  MoveL 657 to (55.18, -49.67, -189.83) mm, rotated rx 42.04 ry 15.1 rz 65.25 deg; joints [-16.317, -43.743, 106.759, 144.666, 49.492, -27.824, -175]
  MoveL 658 to (55.66, -49.78, -189.81) mm, rotated rx 42.04 ry 15.1 rz 65.25 deg; joints [-16.315, -43.768, 106.758, 144.655, 49.471, -27.806, -175]
  MoveL 659 to (56.16, -49.9, -189.79) mm, rotated rx 42.04 ry 15.1 rz 65.25 deg; joints [-16.314, -43.794, 106.756, 144.643, 49.448, -27.785, -175]
  MoveL 660 to (58.7, -50.57, -189.79) mm, rotated rx 42.04 ry 15.1 rz 65.25 deg; joints [-16.31, -43.921, 106.741, 144.577, 49.331, -27.679, -175]
  MoveL 661 to (60.09, -51.01, -189.88) mm, rotated rx 42.04 ry 15.1 rz 65.25 deg; joints [-16.311, -43.987, 106.725, 144.535, 49.264, -27.616, -175]
  MoveL 662 to (61.18, -51.5, -190.13) mm, rotated rx 42.04 ry 15.1 rz 65.25 deg; joints [-16.317, -44.033, 106.696, 144.49, 49.205, -27.555, -175]
  MoveL 663 to (61.98, -52.04, -190.54) mm, rotated rx 42.04 ry 15.1 rz 65.25 deg; joints [-16.329, -44.058, 106.654, 144.442, 49.153, -27.497, -175]
  MoveL 664 to (62.49, -52.65, -191.13) mm, rotated rx 42.04 ry 15.1 rz 65.25 deg; joints [-16.347, -44.062, 106.598, 144.39, 49.109, -27.442, -175]
  MoveL 665 to (62.7, -53.31, -191.87) mm, rotated rx 42.04 ry 15.1 rz 65.25 deg; joints [-16.37, -44.047, 106.53, 144.335, 49.073, -27.39, -175]
  MoveL 666 to (62.62, -54.02, -192.79) mm, rotated rx 42.04 ry 15.1 rz 65.25 deg; joints [-16.399, -44.01, 106.448, 144.277, 49.044, -27.341, -175]
  MoveL 667 to (61.57, -55.63, -195.12) mm, rotated rx 42.04 ry 15.1 rz 65.25 deg; joints [-16.475, -43.877, 106.246, 144.15, 49.009, -27.25, -175]
  MoveL 668 to (59.76, -57.01, -197.47) mm, rotated rx 42.04 ry 15.1 rz 65.25 deg; joints [-16.552, -43.706, 106.05, 144.044, 49.009, -27.192, -175]
  MoveL 669 to (57.6, -57.72, -199.17) mm, rotated rx 42.04 ry 15.1 rz 65.25 deg; joints [-16.61, -43.543, 105.918, 143.99, 49.051, -27.188, -175]
  MoveL 670 to (56.4, -57.82, -199.79) mm, rotated rx 42.04 ry 15.1 rz 65.25 deg; joints [-16.631, -43.464, 105.877, 143.983, 49.087, -27.206, -175]
  MoveL 671 to (55.1, -57.75, -200.24) mm, rotated rx 42.04 ry 15.1 rz 65.25 deg; joints [-16.648, -43.387, 105.852, 143.989, 49.134, -27.238, -175]
  MoveL 672 to (52.26, -57.11, -200.67) mm, rotated rx 42.04 ry 15.1 rz 65.25 deg; joints [-16.668, -43.239, 105.851, 144.039, 49.258, -27.343, -175]
  MoveL 673 to (51.3, -56.8, -200.71) mm, rotated rx 42.04 ry 15.1 rz 65.25 deg; joints [-16.672, -43.193, 105.861, 144.063, 49.304, -27.384, -175]
  MoveL 674 to (48.87, -55.82, -200.71) mm, rotated rx 42.04 ry 15.1 rz 65.25 deg; joints [-16.678, -43.084, 105.904, 144.132, 49.429, -27.499, -175]
  MoveL 675 to (47.92, -55.48, -200.77) mm, rotated rx 42.04 ry 15.1 rz 65.25 deg; joints [-16.683, -43.039, 105.916, 144.155, 49.476, -27.541, -175]
  MoveL 676 to (46.95, -55.09, -200.77) mm, rotated rx 42.04 ry 15.1 rz 65.25 deg; joints [-16.685, -42.995, 105.934, 144.183, 49.527, -27.587, -175]
  MoveL 677 to (46.5, -54.91, -200.78) mm, rotated rx 42.04 ry 15.1 rz 65.25 deg; joints [-16.687, -42.974, 105.941, 144.195, 49.55, -27.607, -175]
  MoveL 678 to (46.09, -54.77, -200.8) mm, rotated rx 42.04 ry 15.1 rz 65.25 deg; joints [-16.688, -42.955, 105.946, 144.205, 49.57, -27.625, -175]
  MoveL 679 to (45.66, -54.6, -200.81) mm, rotated rx 42.04 ry 15.1 rz 65.25 deg; joints [-16.69, -42.935, 105.952, 144.216, 49.592, -27.645, -175]
  MoveL 680 to (43.23, -53.62, -200.82) mm, rotated rx 42.04 ry 15.1 rz 65.25 deg; joints [-16.697, -42.825, 105.994, 144.283, 49.717, -27.758, -175]
  MoveL 681 to (42.77, -53.45, -200.83) mm, rotated rx 42.04 ry 15.1 rz 65.25 deg; joints [-16.699, -42.803, 106, 144.295, 49.74, -27.778, -175]
  MoveL 682 to (42.32, -53.31, -200.87) mm, rotated rx 42.04 ry 15.1 rz 65.25 deg; joints [-16.701, -42.781, 106.003, 144.305, 49.761, -27.797, -175]
  MoveL 683 to (41.9, -53.22, -200.91) mm, rotated rx 42.04 ry 15.1 rz 65.25 deg; joints [-16.703, -42.759, 106.003, 144.313, 49.78, -27.812, -175]
  MoveL 684 to (41.47, -53.15, -200.95) mm, rotated rx 42.04 ry 15.1 rz 65.25 deg; joints [-16.705, -42.735, 106.001, 144.321, 49.797, -27.827, -175]
  MoveL 685 to (41.03, -53.15, -200.96) mm, rotated rx 42.04 ry 15.1 rz 65.25 deg; joints [-16.705, -42.709, 105.992, 144.33, 49.811, -27.841, -175]
  MoveL 686 to (40.58, -53.2, -200.97) mm, rotated rx 42.04 ry 15.1 rz 65.25 deg; joints [-16.704, -42.682, 105.98, 144.338, 49.824, -27.852, -175]
  MoveL 687 to (41.34, -53.26, -201.71) mm, rotated rx 42.04 ry 15.1 rz 65.25 deg; joints [-16.732, -42.719, 105.975, 144.283, 49.797, -27.807, -175]
  MoveL 688 to (40.01, -53.79, -202.26) mm, rotated rx 42.04 ry 15.1 rz 65.25 deg; joints [-16.748, -42.619, 105.893, 144.273, 49.816, -27.813, -175]
  MoveL 689 to (38.53, -54.28, -202.68) mm, rotated rx 42.04 ry 15.1 rz 65.25 deg; joints [-16.759, -42.512, 105.814, 144.274, 49.841, -27.829, -175]
  MoveL 690 to (36.83, -54.75, -202.99) mm, rotated rx 42.04 ry 15.1 rz 65.25 deg; joints [-16.766, -42.394, 105.735, 144.285, 49.875, -27.856, -175]
  MoveL 691 to (34.86, -55.21, -203.17) mm, rotated rx 42.04 ry 15.1 rz 65.25 deg; joints [-16.768, -42.262, 105.654, 144.307, 49.917, -27.894, -175]
  MoveL 692 to (32.82, -55.68, -203.37) mm, rotated rx 42.04 ry 15.1 rz 65.25 deg; joints [-16.771, -42.125, 105.57, 144.331, 49.961, -27.934, -175]
  MoveL 693 to (30.73, -56.13, -203.49) mm, rotated rx 42.04 ry 15.1 rz 65.25 deg; joints [-16.77, -41.986, 105.488, 144.359, 50.007, -27.977, -175]
  MoveL 694 to (28.65, -56.6, -203.71) mm, rotated rx 42.04 ry 15.1 rz 65.25 deg; joints [-16.774, -41.847, 105.403, 144.381, 50.051, -28.016, -175]
  MoveL 695 to (26.56, -57.04, -203.83) mm, rotated rx 42.04 ry 15.1 rz 65.25 deg; joints [-16.773, -41.708, 105.321, 144.41, 50.097, -28.059, -175]
  MoveL 696 to (24.48, -57.49, -203.95) mm, rotated rx 42.04 ry 15.1 rz 65.25 deg; joints [-16.773, -41.57, 105.238, 144.437, 50.142, -28.102, -175]
  MoveL 697 to (22.39, -57.93, -204.06) mm, rotated rx 42.04 ry 15.1 rz 65.25 deg; joints [-16.772, -41.432, 105.156, 144.465, 50.188, -28.144, -175]
  MoveL 698 to (20.3, -58.38, -204.3) mm, rotated rx 42.04 ry 15.1 rz 65.25 deg; joints [-16.776, -41.292, 105.071, 144.486, 50.233, -28.183, -175]
  MoveL 699 to (18.21, -58.81, -204.42) mm, rotated rx 42.04 ry 15.1 rz 65.25 deg; joints [-16.776, -41.154, 104.988, 144.514, 50.278, -28.225, -175]
  MoveL 700 to (16.22, -59.29, -204.52) mm, rotated rx 42.04 ry 15.1 rz 65.25 deg; joints [-16.774, -41.02, 104.903, 144.539, 50.317, -28.263, -175]
  MoveL 701 to (14.29, -59.87, -204.73) mm, rotated rx 42.04 ry 15.1 rz 65.25 deg; joints [-16.776, -40.886, 104.809, 144.556, 50.35, -28.292, -175]
  MoveL 702 to (11.83, -60.35, -204.87) mm, rotated rx 42.04 ry 15.1 rz 65.25 deg; joints [-16.776, -40.724, 104.713, 144.587, 50.404, -28.342, -175]
  MoveL 703 to (9.41, -60.7, -204.95) mm, rotated rx 42.04 ry 15.1 rz 65.25 deg; joints [-16.775, -40.569, 104.63, 144.623, 50.462, -28.396, -175]
  MoveL 704 to (7.15, -61.09, -204.98) mm, rotated rx 42.04 ry 15.1 rz 65.25 deg; joints [-16.772, -40.423, 104.547, 144.658, 50.513, -28.446, -175]
  MoveL 705 to (5.14, -61.5, -205.03) mm, rotated rx 42.04 ry 15.1 rz 65.25 deg; joints [-16.769, -40.291, 104.469, 144.686, 50.556, -28.487, -175]
  MoveL 706 to (3.22, -61.89, -205.15) mm, rotated rx 42.04 ry 15.1 rz 65.25 deg; joints [-16.769, -40.164, 104.391, 144.71, 50.596, -28.524, -175]
  MoveL 707 to (1.23, -62.3, -205.21) mm, rotated rx 42.04 ry 15.1 rz 65.25 deg; joints [-16.767, -40.033, 104.311, 144.736, 50.637, -28.563, -175]
  MoveL 708 to (-0.85, -62.72, -205.28) mm, rotated rx 42.04 ry 15.1 rz 65.25 deg; joints [-16.765, -39.896, 104.227, 144.764, 50.681, -28.604, -175]
  MoveL 709 to (-2.8, -63.09, -205.46) mm, rotated rx 42.04 ry 15.1 rz 65.25 deg; joints [-16.767, -39.767, 104.148, 144.784, 50.722, -28.64, -175]
  MoveL 710 to (-4.68, -63.43, -205.78) mm, rotated rx 42.04 ry 15.1 rz 65.25 deg; joints [-16.775, -39.643, 104.071, 144.797, 50.763, -28.671, -175]
  MoveL 711 to (-5.49, -63.13, -206.82) mm, rotated rx 42.04 ry 15.1 rz 65.25 deg; joints [-16.816, -39.595, 104.059, 144.765, 50.801, -28.679, -175]
  MoveL 712 to (-5.26, -63.03, -207.34) mm, rotated rx 42.04 ry 15.1 rz 65.25 deg; joints [-16.837, -39.609, 104.063, 144.736, 50.799, -28.663, -175]
  MoveL 713 to (-5.25, -63, -207.66) mm, rotated rx 42.04 ry 15.1 rz 65.25 deg; joints [-16.849, -39.607, 104.059, 144.72, 50.8, -28.655, -175]
  MoveL 714 to (-5.46, -63.06, -207.82) mm, rotated rx 42.04 ry 15.1 rz 65.25 deg; joints [-16.855, -39.592, 104.046, 144.715, 50.804, -28.654, -175]
  MoveL 715 to (-5.84, -63.24, -207.86) mm, rotated rx 42.04 ry 15.1 rz 65.25 deg; joints [-16.854, -39.563, 104.021, 144.717, 50.806, -28.657, -175]
  MoveL 716 to (-6.28, -63.52, -207.87) mm, rotated rx 42.04 ry 15.1 rz 65.25 deg; joints [-16.852, -39.528, 103.986, 144.72, 50.806, -28.658, -175]
  MoveL 717 to (-6.74, -63.9, -207.89) mm, rotated rx 42.04 ry 15.1 rz 65.25 deg; joints [-16.849, -39.489, 103.942, 144.721, 50.802, -28.656, -175]
  MoveL 718 to (-7.21, -64.32, -207.9) mm, rotated rx 42.04 ry 15.1 rz 65.25 deg; joints [-16.846, -39.448, 103.895, 144.722, 50.795, -28.652, -175]
  MoveL 719 to (-9.77, -66.94, -207.9) mm, rotated rx 42.04 ry 15.1 rz 65.25 deg; joints [-16.823, -39.214, 103.605, 144.723, 50.745, -28.622, -175]
  MoveL 720 to (-10.09, -67.25, -207.92) mm, rotated rx 42.04 ry 15.1 rz 65.25 deg; joints [-16.822, -39.185, 103.571, 144.722, 50.74, -28.618, -175]
  MoveL 721 to (-10.43, -67.59, -207.93) mm, rotated rx 42.04 ry 15.1 rz 65.25 deg; joints [-16.819, -39.154, 103.532, 144.722, 50.733, -28.614, -175]
  MoveL 722 to (-10.8, -67.96, -207.94) mm, rotated rx 42.04 ry 15.1 rz 65.25 deg; joints [-16.816, -39.12, 103.491, 144.722, 50.726, -28.61, -175]
  MoveL 723 to (-11.16, -68.3, -207.96) mm, rotated rx 42.04 ry 15.1 rz 65.25 deg; joints [-16.814, -39.088, 103.453, 144.721, 50.72, -28.606, -175]
  MoveL 724 to (-11.5, -68.61, -208) mm, rotated rx 42.04 ry 15.1 rz 65.25 deg; joints [-16.812, -39.058, 103.416, 144.72, 50.715, -28.602, -175]
  MoveL 725 to (-11.83, -68.89, -208.06) mm, rotated rx 42.04 ry 15.1 rz 65.25 deg; joints [-16.812, -39.029, 103.383, 144.719, 50.711, -28.599, -175]
  MoveL 726 to (-12.18, -69.21, -208.09) mm, rotated rx 42.04 ry 15.1 rz 65.25 deg; joints [-16.811, -38.998, 103.346, 144.718, 50.706, -28.595, -175]
  MoveL 727 to (-12.53, -69.55, -208.11) mm, rotated rx 42.04 ry 15.1 rz 65.25 deg; joints [-16.808, -38.967, 103.308, 144.717, 50.7, -28.591, -175]
  MoveL 728 to (-12.88, -69.9, -208.11) mm, rotated rx 42.04 ry 15.1 rz 65.25 deg; joints [-16.805, -38.934, 103.268, 144.717, 50.693, -28.587, -175]
  MoveL 729 to (-13.25, -70.28, -208.11) mm, rotated rx 42.04 ry 15.1 rz 65.25 deg; joints [-16.802, -38.901, 103.227, 144.717, 50.686, -28.583, -175]
  MoveL 730 to (-15.49, -72.15, -208.46) mm, rotated rx 42.04 ry 15.1 rz 65.25 deg; joints [-16.798, -38.707, 103.002, 144.707, 50.66, -28.562, -175]
  MoveL 731 to (-16.62, -72.79, -208.89) mm, rotated rx 42.04 ry 15.1 rz 65.25 deg; joints [-16.809, -38.616, 102.911, 144.694, 50.662, -28.556, -175]
  MoveL 732 to (-17.76, -73.23, -209.5) mm, rotated rx 42.04 ry 15.1 rz 65.25 deg; joints [-16.827, -38.53, 102.834, 144.677, 50.674, -28.555, -175]
  MoveL 733 to (-20.07, -73.52, -211.23) mm, rotated rx 42.04 ry 15.1 rz 65.25 deg; joints [-16.888, -38.371, 102.72, 144.626, 50.726, -28.561, -175]
  MoveL 734 to (-22.42, -73.02, -213.65) mm, rotated rx 42.04 ry 15.1 rz 65.25 deg; joints [-16.981, -38.228, 102.662, 144.555, 50.818, -28.581, -175]
  MoveL 735 to (-24.17, -71.99, -216.08) mm, rotated rx 42.04 ry 15.1 rz 65.25 deg; joints [-17.078, -38.138, 102.663, 144.483, 50.918, -28.607, -175]
  MoveL 736 to (-24.6, -71.37, -217.03) mm, rotated rx 42.04 ry 15.1 rz 65.25 deg; joints [-17.119, -38.124, 102.689, 144.454, 50.96, -28.618, -175]
  MoveL 737 to (-24.72, -70.69, -217.81) mm, rotated rx 42.04 ry 15.1 rz 65.25 deg; joints [-17.153, -38.132, 102.731, 144.429, 50.996, -28.628, -175]
  MoveL 738 to (-24.66, -70.32, -218.13) mm, rotated rx 42.04 ry 15.1 rz 65.25 deg; joints [-17.168, -38.144, 102.759, 144.418, 51.012, -28.632, -175]
  MoveL 739 to (-24.53, -69.94, -218.41) mm, rotated rx 42.04 ry 15.1 rz 65.25 deg; joints [-17.182, -38.162, 102.79, 144.408, 51.027, -28.637, -175]
  MoveL 740 to (-24.05, -69.12, -218.84) mm, rotated rx 42.04 ry 15.1 rz 65.25 deg; joints [-17.205, -38.212, 102.865, 144.392, 51.053, -28.645, -175]
  MoveL 741 to (-23.26, -68.24, -219.1) mm, rotated rx 42.04 ry 15.1 rz 65.25 deg; joints [-17.223, -38.285, 102.957, 144.38, 51.073, -28.651, -175]
  MoveL 742 to (-22.17, -67.28, -219.19) mm, rotated rx 42.04 ry 15.1 rz 65.25 deg; joints [-17.235, -38.379, 103.065, 144.373, 51.088, -28.657, -175]
  MoveL 743 to (-21.76, -66.96, -219.19) mm, rotated rx 42.04 ry 15.1 rz 65.25 deg; joints [-17.238, -38.413, 103.104, 144.371, 51.092, -28.658, -175]
  MoveL 744 to (-21.39, -66.69, -219.16) mm, rotated rx 42.04 ry 15.1 rz 65.25 deg; joints [-17.239, -38.444, 103.137, 144.371, 51.094, -28.66, -175]
  MoveL 745 to (-21.03, -66.45, -219.12) mm, rotated rx 42.04 ry 15.1 rz 65.25 deg; joints [-17.24, -38.473, 103.167, 144.371, 51.095, -28.66, -175]
  MoveL 746 to (-20.67, -66.23, -219.06) mm, rotated rx 42.04 ry 15.1 rz 65.25 deg; joints [-17.24, -38.501, 103.197, 144.371, 51.096, -28.661, -175]
  MoveL 747 to (-20.3, -65.97, -219.02) mm, rotated rx 42.04 ry 15.1 rz 65.25 deg; joints [-17.241, -38.532, 103.229, 144.371, 51.098, -28.662, -175]
  MoveL 748 to (-19.89, -65.66, -219) mm, rotated rx 42.04 ry 15.1 rz 65.25 deg; joints [-17.243, -38.566, 103.266, 144.37, 51.101, -28.663, -175]
  MoveL 749 to (-19.48, -65.34, -219) mm, rotated rx 42.04 ry 15.1 rz 65.25 deg; joints [-17.246, -38.6, 103.304, 144.368, 51.105, -28.665, -175]
  MoveL 750 to (-19.09, -65.03, -218.99) mm, rotated rx 42.04 ry 15.1 rz 65.25 deg; joints [-17.249, -38.633, 103.341, 144.367, 51.108, -28.666, -175]
  MoveL 751 to (-18.71, -64.75, -218.97) mm, rotated rx 42.04 ry 15.1 rz 65.25 deg; joints [-17.25, -38.664, 103.375, 144.366, 51.111, -28.668, -175]
  MoveL 752 to (-18.36, -64.5, -218.92) mm, rotated rx 42.04 ry 15.1 rz 65.25 deg; joints [-17.251, -38.693, 103.405, 144.367, 51.112, -28.669, -175]
  MoveL 753 to (-18.01, -64.27, -218.86) mm, rotated rx 42.04 ry 15.1 rz 65.25 deg; joints [-17.251, -38.722, 103.435, 144.367, 51.113, -28.67, -175]
  MoveL 754 to (-17.62, -64.01, -218.8) mm, rotated rx 42.04 ry 15.1 rz 65.25 deg; joints [-17.251, -38.753, 103.469, 144.368, 51.115, -28.671, -175]
  MoveL 755 to (-17.13, -63.65, -218.77) mm, rotated rx 42.04 ry 15.1 rz 65.25 deg; joints [-17.253, -38.794, 103.513, 144.367, 51.118, -28.672, -175]
  MoveL 756 to (-16.49, -63.18, -218.75) mm, rotated rx 42.04 ry 15.1 rz 65.25 deg; joints [-17.256, -38.847, 103.569, 144.364, 51.122, -28.674, -175]
  MoveL 757 to (-15.26, -62.2, -218.75) mm, rotated rx 42.04 ry 15.1 rz 65.25 deg; joints [-17.266, -38.95, 103.683, 144.359, 51.133, -28.678, -175]
  MoveL 758 to (-14.6, -61.7, -218.71) mm, rotated rx 42.04 ry 15.1 rz 65.25 deg; joints [-17.269, -39.006, 103.744, 144.357, 51.138, -28.68, -175]
  MoveL 759 to (-14.1, -61.32, -218.7) mm, rotated rx 42.04 ry 15.1 rz 65.25 deg; joints [-17.272, -39.047, 103.789, 144.355, 51.142, -28.681, -175]
  MoveL 760 to (-13.68, -61.05, -218.7) mm, rotated rx 42.04 ry 15.1 rz 65.25 deg; joints [-17.274, -39.08, 103.822, 144.352, 51.142, -28.68, -175]
  MoveL 761 to (-13.31, -60.86, -218.67) mm, rotated rx 42.04 ry 15.1 rz 65.25 deg; joints [-17.275, -39.108, 103.848, 144.35, 51.141, -28.678, -175]
  MoveL 762 to (-13.11, -60.81, -218.57) mm, rotated rx 42.04 ry 15.1 rz 65.25 deg; joints [-17.272, -39.123, 103.859, 144.353, 51.137, -28.677, -175]
  MoveL 763 to (-13.15, -60.87, -218.35) mm, rotated rx 42.04 ry 15.1 rz 65.25 deg; joints [-17.263, -39.121, 103.857, 144.363, 51.135, -28.681, -175]
  MoveL 764 to (-13.43, -61.05, -218) mm, rotated rx 42.04 ry 15.1 rz 65.25 deg; joints [-17.248, -39.101, 103.842, 144.383, 51.135, -28.691, -175]
  MoveL 765 to (-12.78, -61.49, -217.3) mm, rotated rx 42.04 ry 15.1 rz 65.25 deg; joints [-17.219, -39.131, 103.832, 144.399, 51.095, -28.675, -175]
  MoveL 766 to (-10.78, -61.37, -217.14) mm, rotated rx 42.04 ry 15.1 rz 65.25 deg; joints [-17.215, -39.255, 103.891, 144.372, 51.041, -28.627, -175]
  MoveL 767 to (-8.86, -61.3, -216.86) mm, rotated rx 42.04 ry 15.1 rz 65.25 deg; joints [-17.207, -39.374, 103.947, 144.353, 50.988, -28.584, -175]
  MoveL 768 to (-6.93, -61.19, -216.59) mm, rotated rx 42.04 ry 15.1 rz 65.25 deg; joints [-17.198, -39.494, 104.004, 144.333, 50.935, -28.541, -175]
  MoveL 769 to (-5, -61.08, -216.32) mm, rotated rx 42.04 ry 15.1 rz 65.25 deg; joints [-17.191, -39.614, 104.062, 144.313, 50.883, -28.498, -175]
  MoveL 770 to (-2.97, -60.96, -216.1) mm, rotated rx 42.04 ry 15.1 rz 65.25 deg; joints [-17.185, -39.74, 104.121, 144.289, 50.827, -28.451, -175]
  MoveL 771 to (-0.85, -60.9, -215.96) mm, rotated rx 42.04 ry 15.1 rz 65.25 deg; joints [-17.181, -39.868, 104.176, 144.258, 50.767, -28.396, -175]
  MoveL 772 to (1.68, -60.93, -215.85) mm, rotated rx 42.04 ry 15.1 rz 65.25 deg; joints [-17.179, -40.018, 104.23, 144.215, 50.688, -28.325, -175]
  MoveL 773 to (4.15, -60.61, -215.78) mm, rotated rx 42.04 ry 15.1 rz 65.25 deg; joints [-17.18, -40.175, 104.313, 144.178, 50.629, -28.269, -175]
  MoveL 774 to (6.25, -60.33, -215.66) mm, rotated rx 42.04 ry 15.1 rz 65.25 deg; joints [-17.179, -40.309, 104.384, 144.148, 50.578, -28.222, -175]
  MoveL 775 to (8.13, -60.14, -215.48) mm, rotated rx 42.04 ry 15.1 rz 65.25 deg; joints [-17.176, -40.428, 104.445, 144.125, 50.529, -28.179, -175]
  MoveL 776 to (10.16, -59.96, -215.36) mm, rotated rx 42.04 ry 15.1 rz 65.25 deg; joints [-17.174, -40.554, 104.505, 144.095, 50.475, -28.13, -175]
  MoveL 777 to (12.24, -59.79, -215.22) mm, rotated rx 42.04 ry 15.1 rz 65.25 deg; joints [-17.171, -40.683, 104.566, 144.065, 50.419, -28.079, -175]
  MoveL 778 to (14.4, -59.62, -215.16) mm, rotated rx 42.04 ry 15.1 rz 65.25 deg; joints [-17.172, -40.817, 104.627, 144.029, 50.361, -28.023, -175]
  MoveL 779 to (16.53, -59.44, -214.93) mm, rotated rx 42.04 ry 15.1 rz 65.25 deg; joints [-17.166, -40.95, 104.691, 144.002, 50.303, -27.973, -175]
  MoveL 780 to (18.66, -59.26, -214.82) mm, rotated rx 42.04 ry 15.1 rz 65.25 deg; joints [-17.165, -41.082, 104.752, 143.969, 50.245, -27.919, -175]
  MoveL 781 to (20.78, -59.07, -214.6) mm, rotated rx 42.04 ry 15.1 rz 65.25 deg; joints [-17.159, -41.216, 104.816, 143.942, 50.188, -27.869, -175]
  MoveL 782 to (22.91, -58.88, -214.49) mm, rotated rx 42.04 ry 15.1 rz 65.25 deg; joints [-17.158, -41.348, 104.877, 143.908, 50.13, -27.815, -175]
  MoveL 783 to (25.04, -58.68, -214.27) mm, rotated rx 42.04 ry 15.1 rz 65.25 deg; joints [-17.153, -41.481, 104.942, 143.88, 50.073, -27.764, -175]
  MoveL 784 to (27.16, -58.49, -214.16) mm, rotated rx 42.04 ry 15.1 rz 65.25 deg; joints [-17.152, -41.613, 105.002, 143.846, 50.015, -27.71, -175]
  MoveL 785 to (29.29, -58.3, -214.05) mm, rotated rx 42.04 ry 15.1 rz 65.25 deg; joints [-17.151, -41.745, 105.062, 143.812, 49.957, -27.655, -175]
  MoveL 786 to (31.19, -58.06, -213.82) mm, rotated rx 42.04 ry 15.1 rz 65.25 deg; joints [-17.145, -41.866, 105.124, 143.789, 49.907, -27.612, -175]
  MoveL 787 to (33, -57.8, -213.52) mm, rotated rx 42.04 ry 15.1 rz 65.25 deg; joints [-17.137, -41.984, 105.188, 143.772, 49.862, -27.574, -175]
  MoveL 788 to (34.78, -57.5, -213.13) mm, rotated rx 42.04 ry 15.1 rz 65.25 deg; joints [-17.126, -42.101, 105.256, 143.761, 49.819, -27.541, -175]
  MoveL 789 to (33.37, -57.33, -212.2) mm, rotated rx 42.04 ry 15.1 rz 65.25 deg; joints [-17.092, -42.031, 105.262, 143.84, 49.871, -27.616, -175]
  MoveL 790 to (33.73, -57.31, -212.15) mm, rotated rx 42.04 ry 15.1 rz 65.25 deg; joints [-17.09, -42.054, 105.272, 143.836, 49.861, -27.607, -175]
  MoveL 791 to (34.1, -57.32, -212.09) mm, rotated rx 42.04 ry 15.1 rz 65.25 deg; joints [-17.088, -42.076, 105.279, 143.831, 49.848, -27.597, -175]
  MoveL 792 to (34.51, -57.41, -212.06) mm, rotated rx 42.04 ry 15.1 rz 65.25 deg; joints [-17.086, -42.097, 105.28, 143.823, 49.831, -27.582, -175]
  MoveL 793 to (34.93, -57.56, -212.03) mm, rotated rx 42.04 ry 15.1 rz 65.25 deg; joints [-17.084, -42.117, 105.275, 143.812, 49.811, -27.564, -175]
  MoveL 794 to (35.39, -57.78, -212.03) mm, rotated rx 42.04 ry 15.1 rz 65.25 deg; joints [-17.082, -42.137, 105.264, 143.8, 49.786, -27.541, -175]
  MoveL 795 to (35.84, -58.02, -212.02) mm, rotated rx 42.04 ry 15.1 rz 65.25 deg; joints [-17.08, -42.155, 105.252, 143.786, 49.76, -27.518, -175]
  MoveL 796 to (36.76, -58.54, -212.02) mm, rotated rx 42.04 ry 15.1 rz 65.25 deg; joints [-17.077, -42.192, 105.224, 143.758, 49.706, -27.469, -175]
  MoveL 797 to (37.19, -58.76, -212) mm, rotated rx 42.04 ry 15.1 rz 65.25 deg; joints [-17.074, -42.21, 105.212, 143.746, 49.682, -27.447, -175]
  MoveL 798 to (37.62, -58.96, -211.95) mm, rotated rx 42.04 ry 15.1 rz 65.25 deg; joints [-17.071, -42.229, 105.204, 143.736, 49.659, -27.428, -175]
  MoveL 799 to (38.1, -59.17, -211.88) mm, rotated rx 42.04 ry 15.1 rz 65.25 deg; joints [-17.067, -42.251, 105.196, 143.727, 49.634, -27.407, -175]
  MoveL 800 to (38.62, -59.42, -211.81) mm, rotated rx 42.04 ry 15.1 rz 65.25 deg; joints [-17.063, -42.274, 105.185, 143.715, 49.605, -27.383, -175]
  MoveL 801 to (39.13, -59.68, -211.78) mm, rotated rx 42.04 ry 15.1 rz 65.25 deg; joints [-17.059, -42.295, 105.172, 143.701, 49.577, -27.357, -175]
  MoveL 802 to (39.61, -59.94, -211.77) mm, rotated rx 42.04 ry 15.1 rz 65.25 deg; joints [-17.057, -42.315, 105.158, 143.687, 49.55, -27.333, -175]
  MoveL 803 to (40.07, -60.2, -211.76) mm, rotated rx 42.04 ry 15.1 rz 65.25 deg; joints [-17.055, -42.333, 105.144, 143.673, 49.522, -27.308, -175]
  MoveL 804 to (40.99, -60.71, -211.76) mm, rotated rx 42.04 ry 15.1 rz 65.25 deg; joints [-17.051, -42.37, 105.115, 143.644, 49.469, -27.259, -175]
  MoveL 805 to (41.9, -61.19, -211.74) mm, rotated rx 42.04 ry 15.1 rz 65.25 deg; joints [-17.047, -42.408, 105.091, 143.618, 49.418, -27.213, -175]
  MoveL 806 to (44.19, -62.47, -211.74) mm, rotated rx 42.04 ry 15.1 rz 65.25 deg; joints [-17.038, -42.498, 105.019, 143.546, 49.285, -27.09, -175]
  MoveL 807 to (45.41, -63.23, -211.83) mm, rotated rx 42.04 ry 15.1 rz 65.25 deg; joints [-17.036, -42.543, 104.972, 143.502, 49.21, -27.019, -175]
  MoveL 808 to (46.33, -63.98, -212.09) mm, rotated rx 42.04 ry 15.1 rz 65.25 deg; joints [-17.04, -42.569, 104.917, 143.455, 49.146, -26.953, -175]
  MoveL 809 to (46.93, -64.7, -212.53) mm, rotated rx 42.04 ry 15.1 rz 65.25 deg; joints [-17.051, -42.576, 104.855, 143.407, 49.094, -26.893, -175]
  MoveL 810 to (47.11, -65.05, -212.81) mm, rotated rx 42.04 ry 15.1 rz 65.25 deg; joints [-17.059, -42.573, 104.821, 143.381, 49.072, -26.866, -175]
  MoveL 811 to (47.22, -65.4, -213.14) mm, rotated rx 42.04 ry 15.1 rz 65.25 deg; joints [-17.068, -42.564, 104.786, 143.356, 49.053, -26.84, -175]
  MoveL 812 to (47.19, -66.08, -213.93) mm, rotated rx 42.04 ry 15.1 rz 65.25 deg; joints [-17.092, -42.533, 104.709, 143.303, 49.023, -26.792, -175]
  MoveL 813 to (46.85, -66.74, -214.9) mm, rotated rx 42.04 ry 15.1 rz 65.25 deg; joints [-17.123, -42.483, 104.625, 143.249, 49.004, -26.75, -175]
  MoveL 814 to (45.24, -68, -217.35) mm, rotated rx 42.04 ry 15.1 rz 65.25 deg; joints [-17.203, -42.326, 104.435, 143.134, 49, -26.684, -175]
  MoveL 815 to (42.96, -68.83, -219.81) mm, rotated rx 42.04 ry 15.1 rz 65.25 deg; joints [-17.287, -42.145, 104.271, 143.042, 49.037, -26.656, -175]
  MoveL 816 to (40.6, -68.88, -221.56) mm, rotated rx 42.04 ry 15.1 rz 65.25 deg; joints [-17.351, -41.991, 104.187, 143.001, 49.111, -26.68, -175]
  MoveL 817 to (39.39, -68.61, -222.18) mm, rotated rx 42.04 ry 15.1 rz 65.25 deg; joints [-17.375, -41.925, 104.176, 143.001, 49.162, -26.712, -175]
  MoveL 818 to (38.16, -68.16, -222.61) mm, rotated rx 42.04 ry 15.1 rz 65.25 deg; joints [-17.394, -41.865, 104.185, 143.013, 49.222, -26.757, -175]
  MoveL 819 to (35.64, -66.66, -222.97) mm, rotated rx 42.04 ry 15.1 rz 65.25 deg; joints [-17.419, -41.766, 104.263, 143.076, 49.371, -26.886, -175]
  MoveL 820 to (33.52, -65.1, -222.96) mm, rotated rx 42.04 ry 15.1 rz 65.25 deg; joints [-17.431, -41.694, 104.362, 143.148, 49.51, -27.014, -175]
  MoveL 821 to (33.1, -64.78, -222.95) mm, rotated rx 42.04 ry 15.1 rz 65.25 deg; joints [-17.433, -41.68, 104.382, 143.164, 49.538, -27.041, -175]
  MoveL 822 to (32.68, -64.44, -222.92) mm, rotated rx 42.04 ry 15.1 rz 65.25 deg; joints [-17.434, -41.667, 104.405, 143.18, 49.567, -27.068, -175]
  MoveL 823 to (32.28, -64.14, -222.91) mm, rotated rx 42.04 ry 15.1 rz 65.25 deg; joints [-17.436, -41.654, 104.424, 143.194, 49.594, -27.093, -175]
  MoveL 824 to (31.92, -63.89, -222.93) mm, rotated rx 42.04 ry 15.1 rz 65.25 deg; joints [-17.439, -41.641, 104.439, 143.205, 49.617, -27.113, -175]
  MoveL 825 to (31.52, -63.61, -222.96) mm, rotated rx 42.04 ry 15.1 rz 65.25 deg; joints [-17.442, -41.626, 104.456, 143.217, 49.643, -27.136, -175]
  MoveL 826 to (31.03, -63.3, -223.02) mm, rotated rx 42.04 ry 15.1 rz 65.25 deg; joints [-17.447, -41.607, 104.472, 143.23, 49.673, -27.162, -175]
  MoveL 827 to (30.53, -63, -223.1) mm, rotated rx 42.04 ry 15.1 rz 65.25 deg; joints [-17.452, -41.588, 104.487, 143.241, 49.702, -27.187, -175]
  MoveL 828 to (30.06, -62.69, -223.15) mm, rotated rx 42.04 ry 15.1 rz 65.25 deg; joints [-17.456, -41.57, 104.505, 143.254, 49.731, -27.212, -175]
  MoveL 829 to (29.62, -62.39, -223.18) mm, rotated rx 42.04 ry 15.1 rz 65.25 deg; joints [-17.459, -41.554, 104.522, 143.267, 49.759, -27.237, -175]
  MoveL 830 to (29.2, -62.09, -223.19) mm, rotated rx 42.04 ry 15.1 rz 65.25 deg; joints [-17.462, -41.539, 104.541, 143.281, 49.787, -27.262, -175]
  MoveL 831 to (28.78, -61.78, -223.19) mm, rotated rx 42.04 ry 15.1 rz 65.25 deg; joints [-17.464, -41.525, 104.56, 143.295, 49.814, -27.287, -175]
  MoveL 832 to (28.31, -61.46, -223.22) mm, rotated rx 42.04 ry 15.1 rz 65.25 deg; joints [-17.468, -41.507, 104.578, 143.309, 49.844, -27.313, -175]
  MoveL 833 to (27.84, -61.17, -223.27) mm, rotated rx 42.04 ry 15.1 rz 65.25 deg; joints [-17.472, -41.489, 104.594, 143.321, 49.872, -27.338, -175]
  MoveL 834 to (27.35, -60.89, -223.34) mm, rotated rx 42.04 ry 15.1 rz 65.25 deg; joints [-17.477, -41.469, 104.607, 143.332, 49.9, -27.362, -175]
  MoveL 835 to (26.89, -60.69, -223.4) mm, rotated rx 42.04 ry 15.1 rz 65.25 deg; joints [-17.48, -41.448, 104.615, 143.342, 49.924, -27.383, -175]
  MoveL 836 to (26.45, -60.54, -223.43) mm, rotated rx 42.04 ry 15.1 rz 65.25 deg; joints [-17.483, -41.427, 104.619, 143.352, 49.945, -27.401, -175]
  MoveL 837 to (26.06, -60.48, -223.44) mm, rotated rx 42.04 ry 15.1 rz 65.25 deg; joints [-17.483, -41.406, 104.617, 143.361, 49.96, -27.416, -175]
  MoveL 838 to (25.67, -60.44, -223.44) mm, rotated rx 42.04 ry 15.1 rz 65.25 deg; joints [-17.483, -41.384, 104.612, 143.369, 49.974, -27.429, -175]
  MoveL 839 to (26.93, -60.72, -224.32) mm, rotated rx 42.04 ry 15.1 rz 65.25 deg; joints [-17.515, -41.441, 104.595, 143.294, 49.922, -27.355, -175]
  MoveL 840 to (25.33, -60.76, -224.6) mm, rotated rx 42.04 ry 15.1 rz 65.25 deg; joints [-17.524, -41.344, 104.554, 143.312, 49.97, -27.395, -175]
  MoveL 841 to (23.52, -60.76, -224.79) mm, rotated rx 42.04 ry 15.1 rz 65.25 deg; joints [-17.53, -41.236, 104.514, 143.338, 50.026, -27.446, -175]
  MoveL 842 to (21.47, -60.71, -224.92) mm, rotated rx 42.04 ry 15.1 rz 65.25 deg; joints [-17.534, -41.117, 104.475, 143.374, 50.092, -27.507, -175]
  MoveL 843 to (19.22, -60.62, -225.01) mm, rotated rx 42.04 ry 15.1 rz 65.25 deg; joints [-17.537, -40.987, 104.436, 143.416, 50.166, -27.576, -175]
  MoveL 844 to (17.09, -60.56, -225.16) mm, rotated rx 42.04 ry 15.1 rz 65.25 deg; joints [-17.541, -40.862, 104.395, 143.452, 50.234, -27.639, -175]
  MoveL 845 to (14.95, -60.51, -225.37) mm, rotated rx 42.04 ry 15.1 rz 65.25 deg; joints [-17.548, -40.736, 104.352, 143.485, 50.303, -27.699, -175]
  MoveL 846 to (12.93, -60.44, -225.5) mm, rotated rx 42.04 ry 15.1 rz 65.25 deg; joints [-17.552, -40.618, 104.314, 143.519, 50.368, -27.759, -175]
  MoveL 847 to (11.08, -60.4, -225.76) mm, rotated rx 42.04 ry 15.1 rz 65.25 deg; joints [-17.561, -40.508, 104.273, 143.543, 50.426, -27.809, -175]
  MoveL 848 to (9.01, -60.34, -225.98) mm, rotated rx 42.04 ry 15.1 rz 65.25 deg; joints [-17.568, -40.387, 104.231, 143.573, 50.492, -27.867, -175]
  MoveL 849 to (6.93, -60.26, -226.12) mm, rotated rx 42.04 ry 15.1 rz 65.25 deg; joints [-17.573, -40.265, 104.192, 143.608, 50.559, -27.928, -175]
  MoveL 850 to (4.8, -60.17, -226.22) mm, rotated rx 42.04 ry 15.1 rz 65.25 deg; joints [-17.576, -40.141, 104.152, 143.645, 50.628, -27.991, -175]
  MoveL 851 to (2.68, -60.09, -226.45) mm, rotated rx 42.04 ry 15.1 rz 65.25 deg; joints [-17.584, -40.016, 104.109, 143.676, 50.696, -28.05, -175]
  MoveL 852 to (0.53, -59.98, -226.71) mm, rotated rx 42.04 ry 15.1 rz 65.25 deg; joints [-17.593, -39.891, 104.067, 143.705, 50.765, -28.11, -175]
  MoveL 853 to (-1.59, -59.88, -226.8) mm, rotated rx 42.04 ry 15.1 rz 65.25 deg; joints [-17.596, -39.768, 104.028, 143.742, 50.834, -28.172, -175]
  MoveL 854 to (-3.76, -59.78, -226.84) mm, rotated rx 42.04 ry 15.1 rz 65.25 deg; joints [-17.597, -39.642, 103.988, 143.783, 50.904, -28.238, -175]
  MoveL 855 to (-5.87, -59.68, -226.95) mm, rotated rx 42.04 ry 15.1 rz 65.25 deg; joints [-17.6, -39.519, 103.949, 143.818, 50.972, -28.299, -175]
  MoveL 856 to (-7.99, -59.57, -227.15) mm, rotated rx 42.04 ry 15.1 rz 65.25 deg; joints [-17.608, -39.396, 103.908, 143.849, 51.04, -28.359, -175]
  MoveL 857 to (-10.06, -59.44, -227.48) mm, rotated rx 42.04 ry 15.1 rz 65.25 deg; joints [-17.62, -39.274, 103.865, 143.873, 51.107, -28.413, -175]
  MoveL 858 to (-12.21, -59.29, -227.74) mm, rotated rx 42.04 ry 15.1 rz 65.25 deg; joints [-17.629, -39.149, 103.824, 143.902, 51.178, -28.473, -175]
  MoveL 859 to (-14.34, -59.15, -227.94) mm, rotated rx 42.04 ry 15.1 rz 65.25 deg; joints [-17.637, -39.025, 103.785, 143.933, 51.247, -28.533, -175]
  MoveL 860 to (-16.51, -58.99, -228.18) mm, rotated rx 42.04 ry 15.1 rz 65.25 deg; joints [-17.645, -38.899, 103.744, 143.962, 51.319, -28.594, -175]
  MoveL 861 to (-18.66, -58.86, -228.32) mm, rotated rx 42.04 ry 15.1 rz 65.25 deg; joints [-17.65, -38.774, 103.703, 143.996, 51.388, -28.655, -175]
  MoveL 862 to (-20.77, -58.76, -228.34) mm, rotated rx 42.04 ry 15.1 rz 65.25 deg; joints [-17.651, -38.651, 103.662, 144.034, 51.454, -28.717, -175]
  MoveL 863 to (-21.27, -58.36, -229.01) mm, rotated rx 42.04 ry 15.1 rz 65.25 deg; joints [-17.679, -38.628, 103.671, 144.016, 51.487, -28.729, -175]
  MoveL 864 to (-20.95, -58.29, -229.34) mm, rotated rx 42.04 ry 15.1 rz 65.25 deg; joints [-17.692, -38.646, 103.678, 143.995, 51.481, -28.714, -175]
  MoveL 865 to (-20.91, -58.28, -229.55) mm, rotated rx 42.04 ry 15.1 rz 65.25 deg; joints [-17.7, -38.648, 103.676, 143.984, 51.481, -28.708, -175]
  MoveL 866 to (-21.12, -58.32, -229.65) mm, rotated rx 42.04 ry 15.1 rz 65.25 deg; joints [-17.703, -38.633, 103.666, 143.982, 51.485, -28.71, -175]
  MoveL 867 to (-21.52, -58.46, -229.67) mm, rotated rx 42.04 ry 15.1 rz 65.25 deg; joints [-17.702, -38.605, 103.643, 143.986, 51.49, -28.715, -175]
  MoveC 868 to (-22.42, -58.93, -229.67) mm, rotated rx 42.04 ry 15.1 rz 65.25 deg; joints [-17.698, -38.536, 103.581, 143.994, 51.493, -28.721, -175] to (-23.29, -59.45, -229.67) mm, rotated rx 42.04 ry 15.1 rz 65.25 deg; joints [-17.692, -38.469, 103.514, 144.001, 51.493, -28.724, -175]
  MoveL 869 to (-23.29, -59.45, -229.67) mm, rotated rx 42.04 ry 15.1 rz 65.25 deg; joints [-17.693, -38.468, 103.514, 144.001, 51.493, -28.724, -175]
  MoveL 870 to (-23.76, -59.72, -229.69) mm, rotated rx 42.04 ry 15.1 rz 65.25 deg; joints [-17.691, -38.432, 103.479, 144.004, 51.493, -28.726, -175]
  MoveL 871 to (-24.24, -59.98, -229.74) mm, rotated rx 42.04 ry 15.1 rz 65.25 deg; joints [-17.69, -38.395, 103.444, 144.005, 51.494, -28.727, -175]
  MoveL 872 to (-24.76, -60.24, -229.81) mm, rotated rx 42.04 ry 15.1 rz 65.25 deg; joints [-17.69, -38.356, 103.407, 144.007, 51.497, -28.729, -175]
  MoveL 873 to (-25.28, -60.53, -229.85) mm, rotated rx 42.04 ry 15.1 rz 65.25 deg; joints [-17.689, -38.316, 103.369, 144.009, 51.498, -28.731, -175]
  MoveL 874 to (-26.33, -61.14, -229.88) mm, rotated rx 42.04 ry 15.1 rz 65.25 deg; joints [-17.683, -38.234, 103.289, 144.016, 51.498, -28.735, -175]
  MoveL 875 to (-26.81, -61.41, -229.91) mm, rotated rx 42.04 ry 15.1 rz 65.25 deg; joints [-17.682, -38.197, 103.253, 144.019, 51.499, -28.737, -175]
  MoveL 876 to (-27.24, -61.61, -229.98) mm, rotated rx 42.04 ry 15.1 rz 65.25 deg; joints [-17.683, -38.164, 103.224, 144.019, 51.501, -28.739, -175]
  MoveL 877 to (-27.64, -61.79, -230.07) mm, rotated rx 42.04 ry 15.1 rz 65.25 deg; joints [-17.684, -38.134, 103.197, 144.019, 51.504, -28.74, -175]
  MoveL 878 to (-28.02, -61.98, -230.13) mm, rotated rx 42.04 ry 15.1 rz 65.25 deg; joints [-17.685, -38.105, 103.17, 144.019, 51.506, -28.742, -175]
  MoveL 879 to (-28.42, -62.19, -230.17) mm, rotated rx 42.04 ry 15.1 rz 65.25 deg; joints [-17.684, -38.075, 103.141, 144.02, 51.507, -28.743, -175]
  MoveL 880 to (-30.66, -63.55, -230.17) mm, rotated rx 42.04 ry 15.1 rz 65.25 deg; joints [-17.671, -37.9, 102.967, 144.037, 51.504, -28.749, -175]
  MoveL 881 to (-33.27, -64.82, -230.52) mm, rotated rx 42.04 ry 15.1 rz 65.25 deg; joints [-17.671, -37.702, 102.784, 144.043, 51.516, -28.76, -175]
  MoveL 882 to (-34.51, -65.18, -230.95) mm, rotated rx 42.04 ry 15.1 rz 65.25 deg; joints [-17.683, -37.614, 102.713, 144.037, 51.533, -28.768, -175]
  MoveL 883 to (-35.69, -65.34, -231.55) mm, rotated rx 42.04 ry 15.1 rz 65.25 deg; joints [-17.703, -37.534, 102.657, 144.025, 51.558, -28.778, -175]
  MoveL 884 to (-36.83, -65.31, -232.33) mm, rotated rx 42.04 ry 15.1 rz 65.25 deg; joints [-17.731, -37.461, 102.615, 144.006, 51.59, -28.789, -175]
  MoveL 885 to (-37.91, -65.1, -233.27) mm, rotated rx 42.04 ry 15.1 rz 65.25 deg; joints [-17.768, -37.395, 102.587, 143.981, 51.63, -28.802, -175]
  MoveL 886 to (-39.94, -64.1, -235.69) mm, rotated rx 42.04 ry 15.1 rz 65.25 deg; joints [-17.865, -37.284, 102.574, 143.912, 51.733, -28.833, -175]
  MoveL 887 to (-41.27, -62.73, -238.1) mm, rotated rx 42.04 ry 15.1 rz 65.25 deg; joints [-17.966, -37.226, 102.61, 143.837, 51.833, -28.86, -175]
  MoveL 888 to (-41.48, -62.06, -239.05) mm, rotated rx 42.04 ry 15.1 rz 65.25 deg; joints [-18.007, -37.226, 102.644, 143.805, 51.871, -28.868, -175]
  MoveL 889 to (-41.39, -61.38, -239.83) mm, rotated rx 42.04 ry 15.1 rz 65.25 deg; joints [-18.041, -37.246, 102.689, 143.776, 51.9, -28.872, -175]
  MoveL 890 to (-41.23, -61.05, -240.15) mm, rotated rx 42.04 ry 15.1 rz 65.25 deg; joints [-18.057, -37.262, 102.715, 143.763, 51.911, -28.873, -175]
  MoveL 891 to (-40.99, -60.72, -240.43) mm, rotated rx 42.04 ry 15.1 rz 65.25 deg; joints [-18.07, -37.284, 102.744, 143.75, 51.921, -28.873, -175]
  MoveL 892 to (-40.3, -60.05, -240.86) mm, rotated rx 42.04 ry 15.1 rz 65.25 deg; joints [-18.093, -37.342, 102.811, 143.728, 51.933, -28.87, -175]
  MoveL 893 to (-39.31, -59.39, -241.12) mm, rotated rx 42.04 ry 15.1 rz 65.25 deg; joints [-18.109, -37.419, 102.888, 143.709, 51.937, -28.863, -175]
  MoveL 894 to (-38.01, -58.73, -241.21) mm, rotated rx 42.04 ry 15.1 rz 65.25 deg; joints [-18.119, -37.516, 102.976, 143.693, 51.933, -28.852, -175]
  MoveL 895 to (-37.53, -58.52, -241.21) mm, rotated rx 42.04 ry 15.1 rz 65.25 deg; joints [-18.121, -37.551, 103.007, 143.689, 51.93, -28.848, -175]
  MoveL 896 to (-37.12, -58.35, -241.17) mm, rotated rx 42.04 ry 15.1 rz 65.25 deg; joints [-18.122, -37.581, 103.033, 143.686, 51.926, -28.844, -175]
  MoveL 897 to (-36.72, -58.21, -241.12) mm, rotated rx 42.04 ry 15.1 rz 65.25 deg; joints [-18.121, -37.609, 103.056, 143.684, 51.922, -28.841, -175]
  MoveL 898 to (-36.33, -58.09, -241.05) mm, rotated rx 42.04 ry 15.1 rz 65.25 deg; joints [-18.12, -37.637, 103.078, 143.683, 51.917, -28.837, -175]
  MoveL 899 to (-35.92, -57.93, -241) mm, rotated rx 42.04 ry 15.1 rz 65.25 deg; joints [-18.12, -37.667, 103.103, 143.681, 51.913, -28.833, -175]
  MoveL 900 to (-35.45, -57.73, -240.98) mm, rotated rx 42.04 ry 15.1 rz 65.25 deg; joints [-18.121, -37.701, 103.132, 143.677, 51.91, -28.829, -175]
  MoveL 901 to (-30.23, -55.38, -240.97) mm, rotated rx 42.04 ry 15.1 rz 65.25 deg; joints [-18.146, -38.084, 103.466, 143.625, 51.876, -28.782, -175]
  MoveL 902 to (-29.53, -55.08, -240.96) mm, rotated rx 42.04 ry 15.1 rz 65.25 deg; joints [-18.149, -38.136, 103.51, 143.618, 51.871, -28.775, -175]
  MoveL 903 to (-28.91, -54.84, -240.95) mm, rotated rx 42.04 ry 15.1 rz 65.25 deg; joints [-18.151, -38.179, 103.545, 143.612, 51.865, -28.767, -175]
  MoveL 904 to (-28.35, -54.72, -240.94) mm, rotated rx 42.04 ry 15.1 rz 65.25 deg; joints [-18.152, -38.217, 103.57, 143.604, 51.854, -28.757, -175]
  MoveL 905 to (-27.81, -54.68, -240.9) mm, rotated rx 42.04 ry 15.1 rz 65.25 deg; joints [-18.151, -38.251, 103.587, 143.598, 51.841, -28.745, -175]
  MoveL 906 to (-27.48, -54.71, -240.74) mm, rotated rx 42.04 ry 15.1 rz 65.25 deg; joints [-18.145, -38.271, 103.595, 143.599, 51.83, -28.739, -175]
  MoveL 907 to (-27.48, -54.74, -240.43) mm, rotated rx 42.04 ry 15.1 rz 65.25 deg; joints [-18.133, -38.272, 103.6, 143.614, 51.829, -28.746, -175]
  MoveL 908 to (-27.85, -54.75, -239.94) mm, rotated rx 42.04 ry 15.1 rz 65.25 deg; joints [-18.115, -38.254, 103.6, 143.645, 51.84, -28.768, -175]
  MoveL 909 to (-27.62, -55.34, -238.97) mm, rotated rx 42.04 ry 15.1 rz 65.25 deg; joints [-18.073, -38.258, 103.576, 143.68, 51.806, -28.764, -175]
  MoveL 910 to (-25.78, -55.69, -238.67) mm, rotated rx 42.04 ry 15.1 rz 65.25 deg; joints [-18.06, -38.36, 103.595, 143.657, 51.737, -28.707, -175]
  MoveL 911 to (-23.85, -56.05, -238.46) mm, rotated rx 42.04 ry 15.1 rz 65.25 deg; joints [-18.051, -38.466, 103.614, 143.627, 51.664, -28.646, -175]
  MoveL 912 to (-21.76, -56.41, -238.34) mm, rotated rx 42.04 ry 15.1 rz 65.25 deg; joints [-18.044, -38.581, 103.633, 143.59, 51.586, -28.576, -175]
  MoveL 913 to (-17.55, -57.12, -238.34) mm, rotated rx 42.04 ry 15.1 rz 65.25 deg; joints [-18.041, -38.81, 103.669, 143.503, 51.43, -28.431, -175]
  MoveL 914 to (-15.59, -57.45, -238.25) mm, rotated rx 42.04 ry 15.1 rz 65.25 deg; joints [-18.036, -38.916, 103.687, 143.466, 51.357, -28.366, -175]
  MoveL 915 to (-13.49, -57.8, -238.25) mm, rotated rx 42.04 ry 15.1 rz 65.25 deg; joints [-18.034, -39.031, 103.704, 143.422, 51.279, -28.292, -175]
  MoveL 916 to (-11.38, -58.25, -238.25) mm, rotated rx 42.04 ry 15.1 rz 65.25 deg; joints [-18.032, -39.142, 103.712, 143.376, 51.195, -28.215, -175]
  MoveL 917 to (-8.9, -58.83, -238.07) mm, rotated rx 42.04 ry 15.1 rz 65.25 deg; joints [-18.022, -39.273, 103.721, 143.329, 51.095, -28.126, -175]
  MoveL 918 to (-6.68, -59.07, -237.84) mm, rotated rx 42.04 ry 15.1 rz 65.25 deg; joints [-18.013, -39.398, 103.755, 143.295, 51.019, -28.059, -175]
  MoveL 919 to (-4.53, -59.33, -237.72) mm, rotated rx 42.04 ry 15.1 rz 65.25 deg; joints [-18.007, -39.519, 103.782, 143.257, 50.942, -27.99, -175]
  MoveL 920 to (-2.42, -59.68, -237.61) mm, rotated rx 42.04 ry 15.1 rz 65.25 deg; joints [-18.002, -39.633, 103.799, 143.216, 50.863, -27.918, -175]
  MoveL 921 to (-0.32, -60.02, -237.4) mm, rotated rx 42.04 ry 15.1 rz 65.25 deg; joints [-17.992, -39.748, 103.819, 143.181, 50.785, -27.848, -175]
  MoveL 922 to (1.79, -60.37, -237.29) mm, rotated rx 42.04 ry 15.1 rz 65.25 deg; joints [-17.986, -39.863, 103.837, 143.14, 50.705, -27.776, -175]
  MoveL 923 to (3.89, -60.71, -237.18) mm, rotated rx 42.04 ry 15.1 rz 65.25 deg; joints [-17.981, -39.977, 103.854, 143.099, 50.626, -27.703, -175]
  MoveL 924 to (6, -61.04, -236.97) mm, rotated rx 42.04 ry 15.1 rz 65.25 deg; joints [-17.971, -40.092, 103.874, 143.063, 50.548, -27.633, -175]
  MoveL 925 to (8.11, -61.38, -236.86) mm, rotated rx 42.04 ry 15.1 rz 65.25 deg; joints [-17.966, -40.206, 103.891, 143.022, 50.468, -27.56, -175]
  MoveL 926 to (10.21, -61.72, -236.76) mm, rotated rx 42.04 ry 15.1 rz 65.25 deg; joints [-17.96, -40.32, 103.907, 142.98, 50.389, -27.486, -175]
  MoveL 927 to (12.32, -62.04, -236.55) mm, rotated rx 42.04 ry 15.1 rz 65.25 deg; joints [-17.951, -40.436, 103.928, 142.943, 50.311, -27.416, -175]
  MoveL 928 to (14.43, -62.37, -236.45) mm, rotated rx 42.04 ry 15.1 rz 65.25 deg; joints [-17.946, -40.55, 103.944, 142.9, 50.231, -27.342, -175]
  MoveL 929 to (16.27, -62.58, -236.19) mm, rotated rx 42.04 ry 15.1 rz 65.25 deg; joints [-17.936, -40.653, 103.968, 142.873, 50.165, -27.284, -175]
  MoveL 930 to (17.93, -62.72, -235.82) mm, rotated rx 42.04 ry 15.1 rz 65.25 deg; joints [-17.922, -40.749, 103.997, 142.855, 50.108, -27.238, -175]
  MoveL 931 to (19.46, -62.77, -235.32) mm, rotated rx 42.04 ry 15.1 rz 65.25 deg; joints [-17.904, -40.841, 104.034, 142.849, 50.06, -27.203, -175]
  MoveL 932 to (18.41, -62.34, -234.48) mm, rotated rx 42.04 ry 15.1 rz 65.25 deg; joints [-17.875, -40.801, 104.069, 142.921, 50.112, -27.276, -175]
  MoveL 933 to (18.73, -62.4, -234.45) mm, rotated rx 42.04 ry 15.1 rz 65.25 deg; joints [-17.874, -40.819, 104.071, 142.915, 50.099, -27.264, -175]
  MoveL 934 to (19.05, -62.49, -234.41) mm, rotated rx 42.04 ry 15.1 rz 65.25 deg; joints [-17.872, -40.835, 104.071, 142.909, 50.085, -27.252, -175]
  MoveL 935 to (19.37, -62.66, -234.35) mm, rotated rx 42.04 ry 15.1 rz 65.25 deg; joints [-17.869, -40.848, 104.063, 142.902, 50.067, -27.237, -175]
  MoveL 936 to (19.71, -62.9, -234.31) mm, rotated rx 42.04 ry 15.1 rz 65.25 deg; joints [-17.865, -40.861, 104.05, 142.893, 50.046, -27.218, -175]
  MoveL 937 to (20.08, -63.21, -234.29) mm, rotated rx 42.04 ry 15.1 rz 65.25 deg; joints [-17.862, -40.873, 104.03, 142.881, 50.02, -27.195, -175]
  MoveL 938 to (23.51, -66.44, -234.29) mm, rotated rx 42.04 ry 15.1 rz 65.25 deg; joints [-17.836, -40.967, 103.812, 142.753, 49.763, -26.96, -175]
  MoveL 939 to (23.82, -66.7, -234.26) mm, rotated rx 42.04 ry 15.1 rz 65.25 deg; joints [-17.833, -40.977, 103.796, 142.744, 49.742, -26.941, -175]
  MoveL 940 to (24.2, -67.06, -234.26) mm, rotated rx 42.04 ry 15.1 rz 65.25 deg; joints [-17.83, -40.987, 103.771, 142.729, 49.714, -26.915, -175]
  MoveL 941 to (24.97, -67.75, -234.22) mm, rotated rx 42.04 ry 15.1 rz 65.25 deg; joints [-17.823, -41.01, 103.726, 142.703, 49.658, -26.865, -175]
  MoveL 942 to (26.87, -69.55, -234.22) mm, rotated rx 42.04 ry 15.1 rz 65.25 deg; joints [-17.808, -41.061, 103.604, 142.631, 49.516, -26.733, -175]
  MoveL 943 to (27.66, -70.21, -234.21) mm, rotated rx 42.04 ry 15.1 rz 65.25 deg; joints [-17.802, -41.085, 103.56, 142.603, 49.461, -26.682, -175]
  MoveL 944 to (28.72, -71.19, -234.27) mm, rotated rx 42.04 ry 15.1 rz 65.25 deg; joints [-17.797, -41.114, 103.493, 142.559, 49.382, -26.608, -175]
  MoveL 945 to (29.48, -72.08, -234.53) mm, rotated rx 42.04 ry 15.1 rz 65.25 deg; joints [-17.799, -41.126, 103.422, 142.513, 49.318, -26.541, -175]
  MoveL 946 to (29.94, -72.89, -234.97) mm, rotated rx 42.04 ry 15.1 rz 65.25 deg; joints [-17.809, -41.121, 103.35, 142.466, 49.266, -26.481, -175]
  MoveL 947 to (30.05, -73.26, -235.26) mm, rotated rx 42.04 ry 15.1 rz 65.25 deg; joints [-17.816, -41.112, 103.312, 142.442, 49.246, -26.455, -175]
  MoveL 948 to (30.09, -73.62, -235.59) mm, rotated rx 42.04 ry 15.1 rz 65.25 deg; joints [-17.826, -41.1, 103.275, 142.417, 49.228, -26.43, -175]
  MoveL 949 to (29.94, -74.26, -236.4) mm, rotated rx 42.04 ry 15.1 rz 65.25 deg; joints [-17.85, -41.062, 103.197, 142.367, 49.204, -26.386, -175]
  MoveL 950 to (29.48, -74.81, -237.4) mm, rotated rx 42.04 ry 15.1 rz 65.25 deg; joints [-17.882, -41.008, 103.117, 142.315, 49.193, -26.349, -175]
  MoveL 951 to (27.66, -75.67, -239.96) mm, rotated rx 42.04 ry 15.1 rz 65.25 deg; joints [-17.968, -40.851, 102.951, 142.207, 49.21, -26.3, -175]
  MoveL 952 to (25.28, -75.96, -242.53) mm, rotated rx 42.04 ry 15.1 rz 65.25 deg; joints [-18.059, -40.68, 102.822, 142.12, 49.269, -26.29, -175]
  MoveL 953 to (23, -75.48, -244.36) mm, rotated rx 42.04 ry 15.1 rz 65.25 deg; joints [-18.129, -40.547, 102.78, 142.084, 49.361, -26.329, -175]
  MoveL 954 to (21.89, -74.94, -245) mm, rotated rx 42.04 ry 15.1 rz 65.25 deg; joints [-18.157, -40.495, 102.792, 142.084, 49.42, -26.368, -175]
  MoveL 955 to (20.81, -74.21, -245.46) mm, rotated rx 42.04 ry 15.1 rz 65.25 deg; joints [-18.18, -40.453, 102.826, 142.097, 49.486, -26.418, -175]
  MoveL 956 to (18.73, -72.17, -245.82) mm, rotated rx 42.04 ry 15.1 rz 65.25 deg; joints [-18.21, -40.396, 102.958, 142.159, 49.644, -26.556, -175]
  MoveL 957 to (16.71, -69.76, -245.82) mm, rotated rx 42.04 ry 15.1 rz 65.25 deg; joints [-18.23, -40.358, 103.132, 142.245, 49.817, -26.717, -175]
  MoveL 958 to (16.04, -68.99, -245.84) mm, rotated rx 42.04 ry 15.1 rz 65.25 deg; joints [-18.237, -40.344, 103.186, 142.272, 49.873, -26.768, -175]
  MoveL 959 to (15.37, -68.19, -245.84) mm, rotated rx 42.04 ry 15.1 rz 65.25 deg; joints [-18.244, -40.331, 103.244, 142.3, 49.93, -26.821, -175]
  MoveL 960 to (15.04, -67.81, -245.84) mm, rotated rx 42.04 ry 15.1 rz 65.25 deg; joints [-18.247, -40.325, 103.271, 142.313, 49.958, -26.846, -175]
  MoveL 961 to (14.61, -67.31, -245.87) mm, rotated rx 42.04 ry 15.1 rz 65.25 deg; joints [-18.253, -40.316, 103.306, 142.33, 49.994, -26.879, -175]
  MoveL 962 to (14.2, -66.87, -245.93) mm, rotated rx 42.04 ry 15.1 rz 65.25 deg; joints [-18.258, -40.306, 103.335, 142.343, 50.027, -26.908, -175]
  MoveL 963 to (13.85, -66.51, -246) mm, rotated rx 42.04 ry 15.1 rz 65.25 deg; joints [-18.264, -40.296, 103.358, 142.353, 50.054, -26.931, -175]
  MoveL 964 to (13.52, -66.18, -246.05) mm, rotated rx 42.04 ry 15.1 rz 65.25 deg; joints [-18.269, -40.287, 103.38, 142.363, 50.08, -26.953, -175]
  MoveL 965 to (13.21, -65.84, -246.08) mm, rotated rx 42.04 ry 15.1 rz 65.25 deg; joints [-18.273, -40.28, 103.403, 142.373, 50.105, -26.975, -175]
  MoveL 966 to (12.2, -64.63, -246.08) mm, rotated rx 42.04 ry 15.1 rz 65.25 deg; joints [-18.283, -40.26, 103.489, 142.415, 50.192, -27.055, -175]
  MoveL 967 to (11.86, -64.26, -246.1) mm, rotated rx 42.04 ry 15.1 rz 65.25 deg; joints [-18.287, -40.252, 103.514, 142.428, 50.219, -27.08, -175]
  MoveL 968 to (11.55, -63.95, -246.13) mm, rotated rx 42.04 ry 15.1 rz 65.25 deg; joints [-18.29, -40.244, 103.535, 142.438, 50.243, -27.101, -175]
  MoveL 969 to (11.26, -63.7, -246.17) mm, rotated rx 42.04 ry 15.1 rz 65.25 deg; joints [-18.294, -40.234, 103.55, 142.446, 50.264, -27.118, -175]
  MoveL 970 to (10.99, -63.56, -246.24) mm, rotated rx 42.04 ry 15.1 rz 65.25 deg; joints [-18.298, -40.222, 103.555, 142.451, 50.278, -27.13, -175]
  MoveL 971 to (10.73, -63.46, -246.31) mm, rotated rx 42.04 ry 15.1 rz 65.25 deg; joints [-18.301, -40.21, 103.557, 142.454, 50.29, -27.14, -175]
  MoveL 972 to (11.92, -64.52, -247.11) mm, rotated rx 42.04 ry 15.1 rz 65.25 deg; joints [-18.322, -40.238, 103.47, 142.371, 50.205, -27.039, -175]
  MoveL 973 to (10.23, -63.99, -247.52) mm, rotated rx 42.04 ry 15.1 rz 65.25 deg; joints [-18.341, -40.153, 103.473, 142.393, 50.28, -27.101, -175]
  MoveL 974 to (8.44, -63.45, -247.78) mm, rotated rx 42.04 ry 15.1 rz 65.25 deg; joints [-18.354, -40.062, 103.477, 142.425, 50.359, -27.17, -175]
  MoveL 975 to (6.51, -62.9, -247.96) mm, rotated rx 42.04 ry 15.1 rz 65.25 deg; joints [-18.364, -39.965, 103.481, 142.464, 50.442, -27.245, -175]
  MoveL 976 to (4.46, -62.34, -248.16) mm, rotated rx 42.04 ry 15.1 rz 65.25 deg; joints [-18.375, -39.861, 103.483, 142.504, 50.529, -27.324, -175]
  MoveL 977 to (2.4, -61.76, -248.25) mm, rotated rx 42.04 ry 15.1 rz 65.25 deg; joints [-18.383, -39.758, 103.489, 142.55, 50.617, -27.406, -175]
  MoveL 978 to (0.35, -61.17, -248.35) mm, rotated rx 42.04 ry 15.1 rz 65.25 deg; joints [-18.39, -39.655, 103.494, 142.595, 50.705, -27.488, -175]
  MoveL 979 to (-1.71, -60.6, -248.55) mm, rotated rx 42.04 ry 15.1 rz 65.25 deg; joints [-18.401, -39.55, 103.496, 142.635, 50.793, -27.566, -175]
  MoveL 980 to (-3.76, -60.01, -248.65) mm, rotated rx 42.04 ry 15.1 rz 65.25 deg; joints [-18.409, -39.447, 103.501, 142.679, 50.881, -27.647, -175]
  MoveL 981 to (-5.81, -59.42, -248.75) mm, rotated rx 42.04 ry 15.1 rz 65.25 deg; joints [-18.416, -39.343, 103.505, 142.723, 50.969, -27.728, -175]
  MoveL 982 to (-7.86, -58.83, -248.95) mm, rotated rx 42.04 ry 15.1 rz 65.25 deg; joints [-18.428, -39.239, 103.507, 142.762, 51.056, -27.806, -175]
  MoveL 983 to (-11.96, -57.64, -249.15) mm, rotated rx 42.04 ry 15.1 rz 65.25 deg; joints [-18.443, -39.032, 103.515, 142.849, 51.232, -27.966, -175]
  MoveL 984 to (-13.68, -57.13, -249.36) mm, rotated rx 42.04 ry 15.1 rz 65.25 deg; joints [-18.454, -38.944, 103.516, 142.879, 51.306, -28.03, -175]
  MoveL 985 to (-15.57, -56.62, -249.43) mm, rotated rx 42.04 ry 15.1 rz 65.25 deg; joints [-18.46, -38.846, 103.516, 142.919, 51.385, -28.103, -175]
  MoveL 986 to (-17.57, -56.14, -249.44) mm, rotated rx 42.04 ry 15.1 rz 65.25 deg; joints [-18.464, -38.742, 103.512, 142.963, 51.466, -28.178, -175]
  MoveL 987 to (-20.13, -55.38, -249.55) mm, rotated rx 42.04 ry 15.1 rz 65.25 deg; joints [-18.473, -38.612, 103.517, 143.016, 51.576, -28.278, -175]
  MoveL 988 to (-22.57, -54.54, -249.64) mm, rotated rx 42.04 ry 15.1 rz 65.25 deg; joints [-18.482, -38.492, 103.532, 143.07, 51.686, -28.378, -175]
  MoveL 989 to (-24.68, -53.87, -249.74) mm, rotated rx 42.04 ry 15.1 rz 65.25 deg; joints [-18.49, -38.386, 103.538, 143.113, 51.778, -28.46, -175]
  MoveL 990 to (-26.64, -53.28, -249.91) mm, rotated rx 42.04 ry 15.1 rz 65.25 deg; joints [-18.501, -38.286, 103.54, 143.149, 51.862, -28.534, -175]
  MoveL 991 to (-28.45, -52.71, -250.19) mm, rotated rx 42.04 ry 15.1 rz 65.25 deg; joints [-18.515, -38.192, 103.54, 143.177, 51.941, -28.599, -175]
  MoveL 992 to (-30.26, -52.15, -250.48) mm, rotated rx 42.04 ry 15.1 rz 65.25 deg; joints [-18.53, -38.099, 103.54, 143.203, 52.019, -28.664, -175]
  MoveL 993 to (-32.04, -51.55, -250.77) mm, rotated rx 42.04 ry 15.1 rz 65.25 deg; joints [-18.545, -38.007, 103.543, 143.229, 52.098, -28.729, -175]
  MoveL 994 to (-33.94, -50.95, -250.93) mm, rotated rx 42.04 ry 15.1 rz 65.25 deg; joints [-18.555, -37.91, 103.545, 143.264, 52.18, -28.8, -175]
  MoveL 995 to (-34.26, -50.38, -251.55) mm, rotated rx 42.04 ry 15.1 rz 65.25 deg; joints [-18.583, -37.903, 103.573, 143.248, 52.216, -28.815, -175]
  MoveL 996 to (-33.95, -50.33, -251.86) mm, rotated rx 42.04 ry 15.1 rz 65.25 deg; joints [-18.595, -37.92, 103.579, 143.228, 52.209, -28.801, -175]
  MoveL 997 to (-33.93, -50.29, -252.05) mm, rotated rx 42.04 ry 15.1 rz 65.25 deg; joints [-18.603, -37.921, 103.579, 143.218, 52.21, -28.797, -175]
  MoveL 998 to (-34.18, -50.27, -252.15) mm, rotated rx 42.04 ry 15.1 rz 65.25 deg; joints [-18.607, -37.906, 103.572, 143.218, 52.218, -28.802, -175]
  MoveL 999 to (-34.62, -50.32, -252.17) mm, rotated rx 42.04 ry 15.1 rz 65.25 deg; joints [-18.606, -37.878, 103.556, 143.224, 52.228, -28.812, -175]
  MoveL 1000 to (-35.1, -50.41, -252.17) mm, rotated rx 42.04 ry 15.1 rz 65.25 deg; joints [-18.605, -37.846, 103.536, 143.231, 52.237, -28.821, -175]
  MoveL 1001 to (-36.04, -50.7, -252.2) mm, rotated rx 42.04 ry 15.1 rz 65.25 deg; joints [-18.603, -37.781, 103.487, 143.241, 52.249, -28.834, -175]
  MoveL 1002 to (-37.53, -51.18, -252.2) mm, rotated rx 42.04 ry 15.1 rz 65.25 deg; joints [-18.598, -37.677, 103.409, 143.259, 52.269, -28.855, -175]
  MoveL 1003 to (-38.48, -51.44, -252.22) mm, rotated rx 42.04 ry 15.1 rz 65.25 deg; joints [-18.595, -37.613, 103.362, 143.27, 52.282, -28.87, -175]
  MoveL 1004 to (-39.48, -51.75, -252.22) mm, rotated rx 42.04 ry 15.1 rz 65.25 deg; joints [-18.591, -37.543, 103.31, 143.283, 52.295, -28.884, -175]
  MoveL 1005 to (-39.97, -51.9, -252.23) mm, rotated rx 42.04 ry 15.1 rz 65.25 deg; joints [-18.59, -37.509, 103.284, 143.288, 52.301, -28.891, -175]
  MoveL 1006 to (-40.42, -52.03, -252.26) mm, rotated rx 42.04 ry 15.1 rz 65.25 deg; joints [-18.59, -37.478, 103.261, 143.292, 52.308, -28.897, -175]
  MoveL 1007 to (-40.85, -52.14, -252.31) mm, rotated rx 42.04 ry 15.1 rz 65.25 deg; joints [-18.59, -37.449, 103.24, 143.295, 52.314, -28.903, -175]
  MoveL 1008 to (-41.24, -52.24, -252.37) mm, rotated rx 42.04 ry 15.1 rz 65.25 deg; joints [-18.591, -37.422, 103.22, 143.297, 52.32, -28.908, -175]
  MoveL 1009 to (-41.65, -52.34, -252.43) mm, rotated rx 42.04 ry 15.1 rz 65.25 deg; joints [-18.592, -37.394, 103.2, 143.3, 52.327, -28.914, -175]
  MoveL 1010 to (-42.09, -52.46, -252.46) mm, rotated rx 42.04 ry 15.1 rz 65.25 deg; joints [-18.592, -37.363, 103.177, 143.304, 52.333, -28.92, -175]
  MoveL 1011 to (-42.55, -52.59, -252.48) mm, rotated rx 42.04 ry 15.1 rz 65.25 deg; joints [-18.591, -37.331, 103.154, 143.308, 52.339, -28.926, -175]
  MoveL 1012 to (-42.98, -52.7, -252.53) mm, rotated rx 42.04 ry 15.1 rz 65.25 deg; joints [-18.591, -37.303, 103.133, 143.312, 52.346, -28.932, -175]
  MoveL 1013 to (-43.37, -52.78, -252.59) mm, rotated rx 42.04 ry 15.1 rz 65.25 deg; joints [-18.593, -37.276, 103.115, 143.314, 52.353, -28.938, -175]
  MoveL 1014 to (-43.77, -52.87, -252.64) mm, rotated rx 42.04 ry 15.1 rz 65.25 deg; joints [-18.593, -37.249, 103.095, 143.317, 52.359, -28.944, -175]
  MoveL 1015 to (-44.2, -52.98, -252.67) mm, rotated rx 42.04 ry 15.1 rz 65.25 deg; joints [-18.593, -37.22, 103.074, 143.321, 52.366, -28.95, -175]
  MoveL 1016 to (-44.7, -53.14, -252.67) mm, rotated rx 42.04 ry 15.1 rz 65.25 deg; joints [-18.591, -37.185, 103.048, 143.327, 52.372, -28.957, -175]
  MoveL 1017 to (-47.54, -53.78, -253.03) mm, rotated rx 42.04 ry 15.1 rz 65.25 deg; joints [-18.597, -36.992, 102.912, 143.347, 52.419, -28.997, -175]
  MoveL 1018 to (-48.83, -53.85, -253.47) mm, rotated rx 42.04 ry 15.1 rz 65.25 deg; joints [-18.611, -36.909, 102.862, 143.345, 52.449, -29.017, -175]
  MoveL 1019 to (-50.03, -53.76, -254.09) mm, rotated rx 42.04 ry 15.1 rz 65.25 deg; joints [-18.634, -36.834, 102.825, 143.335, 52.485, -29.036, -175]
  MoveL 1020 to (-52.15, -53.11, -255.87) mm, rotated rx 42.04 ry 15.1 rz 65.25 deg; joints [-18.705, -36.711, 102.788, 143.293, 52.571, -29.071, -175]
  MoveL 1021 to (-53.9, -51.8, -258.37) mm, rotated rx 42.04 ry 15.1 rz 65.25 deg; joints [-18.809, -36.622, 102.8, 143.219, 52.677, -29.105, -175]
  MoveL 1022 to (-54.89, -50.3, -260.86) mm, rotated rx 42.04 ry 15.1 rz 65.25 deg; joints [-18.915, -36.585, 102.849, 143.135, 52.772, -29.127, -175]
  MoveL 1023 to (-54.95, -49.65, -261.84) mm, rotated rx 42.04 ry 15.1 rz 65.25 deg; joints [-18.957, -36.592, 102.882, 143.097, 52.803, -29.13, -175]
  MoveL 1024 to (-54.71, -49.05, -262.64) mm, rotated rx 42.04 ry 15.1 rz 65.25 deg; joints [-18.993, -36.617, 102.922, 143.063, 52.823, -29.126, -175]
  MoveL 1025 to (-54.48, -48.78, -262.98) mm, rotated rx 42.04 ry 15.1 rz 65.25 deg; joints [-19.008, -36.635, 102.944, 143.047, 52.83, -29.123, -175]
  MoveL 1026 to (-54.18, -48.53, -263.27) mm, rotated rx 42.04 ry 15.1 rz 65.25 deg; joints [-19.021, -36.659, 102.967, 143.032, 52.833, -29.118, -175]
  MoveL 1027 to (-53.36, -48.06, -263.71) mm, rotated rx 42.04 ry 15.1 rz 65.25 deg; joints [-19.043, -36.718, 103.019, 143.003, 52.832, -29.103, -175]
  MoveL 1028 to (-52.24, -47.66, -263.98) mm, rotated rx 42.04 ry 15.1 rz 65.25 deg; joints [-19.058, -36.795, 103.077, 142.977, 52.821, -29.083, -175]
  MoveL 1029 to (-50.83, -47.32, -264.07) mm, rotated rx 42.04 ry 15.1 rz 65.25 deg; joints [-19.065, -36.889, 103.14, 142.955, 52.799, -29.057, -175]
  MoveL 1030 to (-48.26, -46.82, -264.07) mm, rotated rx 42.04 ry 15.1 rz 65.25 deg; joints [-19.072, -37.058, 103.25, 142.919, 52.753, -29.009, -175]
  MoveL 1031 to (-47.82, -46.75, -264.04) mm, rotated rx 42.04 ry 15.1 rz 65.25 deg; joints [-19.072, -37.086, 103.268, 142.915, 52.744, -29.001, -175]
  MoveL 1032 to (-47.42, -46.7, -263.99) mm, rotated rx 42.04 ry 15.1 rz 65.25 deg; joints [-19.071, -37.113, 103.284, 142.911, 52.736, -28.994, -175]
  MoveL 1033 to (-47.04, -46.66, -263.92) mm, rotated rx 42.04 ry 15.1 rz 65.25 deg; joints [-19.069, -37.138, 103.299, 142.909, 52.727, -28.987, -175]
  MoveL 1034 to (-46.61, -46.6, -263.87) mm, rotated rx 42.04 ry 15.1 rz 65.25 deg; joints [-19.068, -37.165, 103.316, 142.905, 52.719, -28.979, -175]
  MoveL 1035 to (-46.12, -46.52, -263.83) mm, rotated rx 42.04 ry 15.1 rz 65.25 deg; joints [-19.068, -37.198, 103.336, 142.9, 52.709, -28.97, -175]
  MoveL 1036 to (-45.6, -46.45, -263.77) mm, rotated rx 42.04 ry 15.1 rz 65.25 deg; joints [-19.067, -37.231, 103.357, 142.895, 52.698, -28.961, -175]
  MoveL 1037 to (-45.06, -46.36, -263.76) mm, rotated rx 42.04 ry 15.1 rz 65.25 deg; joints [-19.067, -37.266, 103.379, 142.888, 52.688, -28.951, -175]
  MoveL 1038 to (-44.43, -46.23, -263.77) mm, rotated rx 42.04 ry 15.1 rz 65.25 deg; joints [-19.07, -37.308, 103.406, 142.879, 52.677, -28.938, -175]
  MoveL 1039 to (-43.59, -46.04, -263.84) mm, rotated rx 42.04 ry 15.1 rz 65.25 deg; joints [-19.075, -37.364, 103.442, 142.864, 52.663, -28.922, -175]
  MoveL 1040 to (-43.07, -45.94, -263.84) mm, rotated rx 42.04 ry 15.1 rz 65.25 deg; joints [-19.076, -37.398, 103.464, 142.857, 52.653, -28.912, -175]
  MoveL 1041 to (-42.58, -45.85, -263.83) mm, rotated rx 42.04 ry 15.1 rz 65.25 deg; joints [-19.077, -37.43, 103.484, 142.85, 52.644, -28.903, -175]
  MoveL 1042 to (-42.12, -45.77, -263.81) mm, rotated rx 42.04 ry 15.1 rz 65.25 deg; joints [-19.077, -37.46, 103.503, 142.845, 52.635, -28.894, -175]
  MoveL 1043 to (-41.71, -45.71, -263.76) mm, rotated rx 42.04 ry 15.1 rz 65.25 deg; joints [-19.076, -37.487, 103.52, 142.841, 52.626, -28.886, -175]
  MoveL 1044 to (-41.31, -45.68, -263.7) mm, rotated rx 42.04 ry 15.1 rz 65.25 deg; joints [-19.075, -37.512, 103.534, 142.838, 52.617, -28.878, -175]
  MoveL 1045 to (-40.89, -45.69, -263.65) mm, rotated rx 42.04 ry 15.1 rz 65.25 deg; joints [-19.073, -37.538, 103.545, 142.833, 52.605, -28.868, -175]
  MoveL 1046 to (-40.48, -45.74, -263.59) mm, rotated rx 42.04 ry 15.1 rz 65.25 deg; joints [-19.071, -37.561, 103.552, 142.828, 52.591, -28.856, -175]
  MoveL 1047 to (-40.27, -45.83, -263.43) mm, rotated rx 42.04 ry 15.1 rz 65.25 deg; joints [-19.064, -37.573, 103.553, 142.831, 52.582, -28.851, -175]
  MoveL 1048 to (-40.37, -45.89, -263.12) mm, rotated rx 42.04 ry 15.1 rz 65.25 deg; joints [-19.052, -37.568, 103.553, 142.847, 52.582, -28.86, -175]
  MoveL 1049 to (-40.81, -45.91, -262.62) mm, rotated rx 42.04 ry 15.1 rz 65.25 deg; joints [-19.033, -37.546, 103.552, 142.879, 52.595, -28.884, -175]
  MoveL 1050 to (-39.98, -46.22, -261.77) mm, rotated rx 42.04 ry 15.1 rz 65.25 deg; joints [-18.999, -37.594, 103.565, 142.902, 52.558, -28.871, -175]
  MoveL 1051 to (-36.04, -47.87, -261.77) mm, rotated rx 42.04 ry 15.1 rz 65.25 deg; joints [-18.986, -37.781, 103.518, 142.809, 52.369, -28.698, -175]
  MoveL 1052 to (-34.2, -48.65, -261.71) mm, rotated rx 42.04 ry 15.1 rz 65.25 deg; joints [-18.978, -37.869, 103.497, 142.768, 52.28, -28.618, -175]
  MoveL 1053 to (-32.37, -49.43, -261.56) mm, rotated rx 42.04 ry 15.1 rz 65.25 deg; joints [-18.966, -37.956, 103.476, 142.73, 52.191, -28.54, -175]
  MoveL 1054 to (-30.26, -50.34, -261.36) mm, rotated rx 42.04 ry 15.1 rz 65.25 deg; joints [-18.952, -38.057, 103.452, 142.689, 52.088, -28.451, -175]
  MoveL 1055 to (-28.27, -51.2, -261.15) mm, rotated rx 42.04 ry 15.1 rz 65.25 deg; joints [-18.937, -38.152, 103.43, 142.65, 51.991, -28.367, -175]
  MoveL 1056 to (-26.26, -52.05, -261.05) mm, rotated rx 42.04 ry 15.1 rz 65.25 deg; joints [-18.927, -38.247, 103.406, 142.605, 51.894, -28.279, -175]
  MoveL 1057 to (-24.29, -52.87, -261.05) mm, rotated rx 42.04 ry 15.1 rz 65.25 deg; joints [-18.921, -38.339, 103.38, 142.557, 51.799, -28.191, -175]
  MoveL 1058 to (-22.46, -53.64, -260.98) mm, rotated rx 42.04 ry 15.1 rz 65.25 deg; joints [-18.912, -38.425, 103.358, 142.514, 51.71, -28.11, -175]
  MoveL 1059 to (-20.73, -54.36, -260.86) mm, rotated rx 42.04 ry 15.1 rz 65.25 deg; joints [-18.903, -38.507, 103.338, 142.477, 51.627, -28.035, -175]
  MoveL 1060 to (-18.84, -55.15, -260.8) mm, rotated rx 42.04 ry 15.1 rz 65.25 deg; joints [-18.894, -38.596, 103.314, 142.432, 51.536, -27.952, -175]
  MoveL 1061 to (-16.87, -55.97, -260.62) mm, rotated rx 42.04 ry 15.1 rz 65.25 deg; joints [-18.881, -38.689, 103.291, 142.391, 51.441, -27.867, -175]
  MoveL 1062 to (-12.93, -57.61, -260.44) mm, rotated rx 42.04 ry 15.1 rz 65.25 deg; joints [-18.862, -38.873, 103.241, 142.299, 51.25, -27.692, -175]
  MoveL 1063 to (-10.96, -58.43, -260.26) mm, rotated rx 42.04 ry 15.1 rz 65.25 deg; joints [-18.849, -38.966, 103.218, 142.258, 51.155, -27.607, -175]
  MoveL 1064 to (-8.98, -59.24, -260.08) mm, rotated rx 42.04 ry 15.1 rz 65.25 deg; joints [-18.836, -39.059, 103.195, 142.215, 51.06, -27.521, -175]
  MoveL 1065 to (-7.02, -60.06, -260.08) mm, rotated rx 42.04 ry 15.1 rz 65.25 deg; joints [-18.83, -39.149, 103.166, 142.164, 50.964, -27.43, -175]
  MoveL 1066 to (-5.04, -60.87, -259.9) mm, rotated rx 42.04 ry 15.1 rz 65.25 deg; joints [-18.817, -39.242, 103.143, 142.121, 50.869, -27.344, -175]
  MoveL 1067 to (-3.06, -61.67, -259.72) mm, rotated rx 42.04 ry 15.1 rz 65.25 deg; joints [-18.805, -39.334, 103.12, 142.077, 50.774, -27.258, -175]
  MoveL 1068 to (-1.09, -62.49, -259.72) mm, rotated rx 42.04 ry 15.1 rz 65.25 deg; joints [-18.799, -39.424, 103.09, 142.025, 50.679, -27.166, -175]
  MoveL 1069 to (0.73, -63.18, -259.53) mm, rotated rx 42.04 ry 15.1 rz 65.25 deg; joints [-18.786, -39.511, 103.073, 141.987, 50.594, -27.089, -175]
  MoveL 1070 to (2.36, -63.72, -259.21) mm, rotated rx 42.04 ry 15.1 rz 65.25 deg; joints [-18.771, -39.592, 103.068, 141.962, 50.521, -27.027, -175]
  MoveL 1071 to (3.83, -64.12, -258.74) mm, rotated rx 42.04 ry 15.1 rz 65.25 deg; joints [-18.751, -39.67, 103.074, 141.949, 50.459, -26.979, -175]
  MoveL 1072 to (3.04, -63.61, -257.98) mm, rotated rx 42.04 ry 15.1 rz 65.25 deg; joints [-18.727, -39.647, 103.121, 142.013, 50.507, -27.045, -175]
  MoveL 1073 to (3.4, -63.81, -257.97) mm, rotated rx 42.04 ry 15.1 rz 65.25 deg; joints [-18.725, -39.662, 103.111, 142.002, 50.487, -27.026, -175]
  MoveC 1074 to (5.59, -66.61, -257.97) mm, rotated rx 42.04 ry 15.1 rz 65.25 deg; joints [-18.701, -39.7, 102.909, 141.909, 50.292, -26.846, -175] to (7.54, -69.58, -257.97) mm, rotated rx 42.04 ry 15.1 rz 65.25 deg; joints [-18.674, -39.717, 102.687, 141.817, 50.096, -26.665, -175]
  MoveL 1075 to (7.54, -69.58, -257.97) mm, rotated rx 42.04 ry 15.1 rz 65.25 deg; joints [-18.674, -39.717, 102.687, 141.817, 50.096, -26.665, -175]
  MoveL 1076 to (7.81, -69.96, -257.95) mm, rotated rx 42.04 ry 15.1 rz 65.25 deg; joints [-18.67, -39.721, 102.658, 141.805, 50.07, -26.642, -175]
  MoveL 1077 to (8.07, -70.3, -257.9) mm, rotated rx 42.04 ry 15.1 rz 65.25 deg; joints [-18.665, -39.725, 102.635, 141.797, 50.047, -26.622, -175]
  MoveL 1078 to (8.32, -70.62, -257.84) mm, rotated rx 42.04 ry 15.1 rz 65.25 deg; joints [-18.66, -39.73, 102.613, 141.789, 50.024, -26.602, -175]
  MoveL 1079 to (8.58, -70.97, -257.79) mm, rotated rx 42.04 ry 15.1 rz 65.25 deg; joints [-18.656, -39.734, 102.589, 141.779, 50, -26.581, -175]
  MoveL 1080 to (8.85, -71.35, -257.76) mm, rotated rx 42.04 ry 15.1 rz 65.25 deg; joints [-18.651, -39.738, 102.561, 141.768, 49.974, -26.558, -175]
  MoveL 1081 to (9.15, -71.78, -257.75) mm, rotated rx 42.04 ry 15.1 rz 65.25 deg; joints [-18.647, -39.741, 102.529, 141.755, 49.946, -26.532, -175]
  MoveL 1082 to (9.72, -72.66, -257.75) mm, rotated rx 42.04 ry 15.1 rz 65.25 deg; joints [-18.639, -39.746, 102.463, 141.728, 49.888, -26.478, -175]
  MoveL 1083 to (10.48, -73.9, -257.84) mm, rotated rx 42.04 ry 15.1 rz 65.25 deg; joints [-18.632, -39.748, 102.366, 141.685, 49.808, -26.401, -175]
  MoveL 1084 to (10.99, -74.99, -258.11) mm, rotated rx 42.04 ry 15.1 rz 65.25 deg; joints [-18.632, -39.739, 102.273, 141.64, 49.742, -26.332, -175]
  MoveL 1085 to (11.26, -75.92, -258.57) mm, rotated rx 42.04 ry 15.1 rz 65.25 deg; joints [-18.641, -39.72, 102.185, 141.594, 49.691, -26.273, -175]
  MoveL 1086 to (11.28, -76.69, -259.21) mm, rotated rx 42.04 ry 15.1 rz 65.25 deg; joints [-18.657, -39.69, 102.102, 141.546, 49.654, -26.222, -175]
  MoveL 1087 to (11.07, -77.3, -260.03) mm, rotated rx 42.04 ry 15.1 rz 65.25 deg; joints [-18.681, -39.649, 102.024, 141.497, 49.632, -26.179, -175]
  MoveL 1088 to (10.62, -77.75, -261.04) mm, rotated rx 42.04 ry 15.1 rz 65.25 deg; joints [-18.714, -39.598, 101.951, 141.447, 49.624, -26.146, -175]
  MoveL 1089 to (8.98, -78.18, -263.6) mm, rotated rx 42.04 ry 15.1 rz 65.25 deg; joints [-18.803, -39.465, 101.82, 141.342, 49.651, -26.105, -175]
  MoveL 1090 to (6.94, -77.93, -266.16) mm, rotated rx 42.04 ry 15.1 rz 65.25 deg; joints [-18.897, -39.331, 101.74, 141.258, 49.721, -26.105, -175]
  MoveL 1091 to (5.99, -77.53, -267.16) mm, rotated rx 42.04 ry 15.1 rz 65.25 deg; joints [-18.937, -39.279, 101.733, 141.234, 49.767, -26.123, -175]
  MoveL 1092 to (5.08, -76.94, -267.99) mm, rotated rx 42.04 ry 15.1 rz 65.25 deg; joints [-18.972, -39.237, 101.746, 141.222, 49.82, -26.152, -175]
  MoveL 1093 to (4.2, -76.17, -268.63) mm, rotated rx 42.04 ry 15.1 rz 65.25 deg; joints [-19.002, -39.206, 101.782, 141.221, 49.881, -26.192, -175]
  MoveL 1094 to (3.37, -75.22, -269.08) mm, rotated rx 42.04 ry 15.1 rz 65.25 deg; joints [-19.027, -39.184, 101.839, 141.233, 49.949, -26.245, -175]
  MoveL 1095 to (1.84, -72.76, -269.45) mm, rotated rx 42.04 ry 15.1 rz 65.25 deg; joints [-19.062, -39.172, 102.016, 141.29, 50.108, -26.383, -175]
  MoveL 1096 to (1.36, -71.83, -269.45) mm, rotated rx 42.04 ry 15.1 rz 65.25 deg; joints [-19.071, -39.174, 102.089, 141.317, 50.165, -26.437, -175]
  MoveL 1097 to (1.12, -71.36, -269.46) mm, rotated rx 42.04 ry 15.1 rz 65.25 deg; joints [-19.075, -39.175, 102.125, 141.33, 50.194, -26.463, -175]
  MoveL 1098 to (0.89, -70.95, -269.48) mm, rotated rx 42.04 ry 15.1 rz 65.25 deg; joints [-19.08, -39.175, 102.157, 141.341, 50.22, -26.487, -175]
  MoveL 1099 to (0.67, -70.58, -269.53) mm, rotated rx 42.04 ry 15.1 rz 65.25 deg; joints [-19.085, -39.174, 102.183, 141.35, 50.243, -26.507, -175]
  MoveL 1100 to (0.46, -70.24, -269.58) mm, rotated rx 42.04 ry 15.1 rz 65.25 deg; joints [-19.09, -39.172, 102.208, 141.357, 50.265, -26.526, -175]
  MoveL 1101 to (0.24, -69.88, -269.63) mm, rotated rx 42.04 ry 15.1 rz 65.25 deg; joints [-19.095, -39.171, 102.234, 141.366, 50.288, -26.546, -175]
  MoveL 1102 to (0.02, -69.47, -269.65) mm, rotated rx 42.04 ry 15.1 rz 65.25 deg; joints [-19.1, -39.171, 102.265, 141.376, 50.314, -26.57, -175]
  MoveL 1103 to (-0.21, -69.03, -269.66) mm, rotated rx 42.04 ry 15.1 rz 65.25 deg; joints [-19.104, -39.172, 102.3, 141.389, 50.341, -26.595, -175]
  MoveL 1104 to (-0.46, -68.53, -269.65) mm, rotated rx 42.04 ry 15.1 rz 65.25 deg; joints [-19.108, -39.173, 102.338, 141.403, 50.371, -26.623, -175]
  MoveL 1105 to (-0.71, -68.06, -269.66) mm, rotated rx 42.04 ry 15.1 rz 65.25 deg; joints [-19.113, -39.174, 102.374, 141.416, 50.4, -26.65, -175]
  MoveL 1106 to (-0.94, -67.63, -269.68) mm, rotated rx 42.04 ry 15.1 rz 65.25 deg; joints [-19.118, -39.174, 102.407, 141.427, 50.427, -26.674, -175]
  MoveL 1107 to (-1.18, -67.22, -269.73) mm, rotated rx 42.04 ry 15.1 rz 65.25 deg; joints [-19.123, -39.173, 102.438, 141.437, 50.453, -26.697, -175]
  MoveL 1108 to (-1.44, -66.79, -269.81) mm, rotated rx 42.04 ry 15.1 rz 65.25 deg; joints [-19.13, -39.171, 102.468, 141.446, 50.481, -26.72, -175]
  MoveL 1109 to (-1.75, -66.27, -269.87) mm, rotated rx 42.04 ry 15.1 rz 65.25 deg; joints [-19.137, -39.168, 102.506, 141.458, 50.514, -26.749, -175]
  MoveL 1110 to (-2.02, -65.77, -269.89) mm, rotated rx 42.04 ry 15.1 rz 65.25 deg; joints [-19.142, -39.168, 102.544, 141.471, 50.546, -26.778, -175]
  MoveL 1111 to (-2.27, -65.3, -269.89) mm, rotated rx 42.04 ry 15.1 rz 65.25 deg; joints [-19.146, -39.169, 102.58, 141.484, 50.574, -26.804, -175]
  MoveL 1112 to (-2.51, -64.83, -269.89) mm, rotated rx 42.04 ry 15.1 rz 65.25 deg; joints [-19.151, -39.17, 102.616, 141.497, 50.603, -26.831, -175]
  MoveL 1113 to (-2.83, -64.26, -269.9) mm, rotated rx 42.04 ry 15.1 rz 65.25 deg; joints [-19.156, -39.17, 102.66, 141.513, 50.639, -26.864, -175]
  MoveL 1114 to (-3.12, -63.75, -269.91) mm, rotated rx 42.04 ry 15.1 rz 65.25 deg; joints [-19.161, -39.168, 102.698, 141.527, 50.671, -26.893, -175]
  MoveL 1115 to (-3.4, -63.33, -269.92) mm, rotated rx 42.04 ry 15.1 rz 65.25 deg; joints [-19.165, -39.165, 102.729, 141.54, 50.699, -26.919, -175]
  MoveL 1116 to (-3.64, -63.08, -269.92) mm, rotated rx 42.04 ry 15.1 rz 65.25 deg; joints [-19.168, -39.159, 102.746, 141.549, 50.718, -26.936, -175]
  MoveL 1117 to (-3.85, -62.92, -269.92) mm, rotated rx 42.04 ry 15.1 rz 65.25 deg; joints [-19.169, -39.152, 102.756, 141.556, 50.732, -26.949, -175]
  MoveL 1118 to (-3.1, -63.48, -270.51) mm, rotated rx 42.04 ry 15.1 rz 65.25 deg; joints [-19.186, -39.172, 102.708, 141.501, 50.683, -26.887, -175]
  MoveL 1119 to (-4.38, -63.09, -271.04) mm, rotated rx 42.04 ry 15.1 rz 65.25 deg; joints [-19.208, -39.105, 102.703, 141.506, 50.738, -26.927, -175]
  MoveL 1120 to (-5.83, -62.49, -271.42) mm, rotated rx 42.04 ry 15.1 rz 65.25 deg; joints [-19.227, -39.035, 102.714, 141.526, 50.806, -26.984, -175]
  MoveL 1121 to (-7.49, -61.69, -271.68) mm, rotated rx 42.04 ry 15.1 rz 65.25 deg; joints [-19.243, -38.961, 102.742, 141.559, 50.891, -27.059, -175]
  MoveL 1122 to (-9.3, -60.72, -271.81) mm, rotated rx 42.04 ry 15.1 rz 65.25 deg; joints [-19.256, -38.883, 102.784, 141.604, 50.988, -27.149, -175]
  MoveL 1123 to (-11.15, -59.72, -271.9) mm, rotated rx 42.04 ry 15.1 rz 65.25 deg; joints [-19.267, -38.805, 102.83, 141.652, 51.088, -27.242, -175]
  MoveL 1124 to (-14.89, -57.67, -272.08) mm, rotated rx 42.04 ry 15.1 rz 65.25 deg; joints [-19.291, -38.647, 102.921, 141.749, 51.29, -27.43, -175]
  MoveL 1125 to (-16.76, -56.65, -272.26) mm, rotated rx 42.04 ry 15.1 rz 65.25 deg; joints [-19.306, -38.566, 102.963, 141.793, 51.391, -27.521, -175]
  MoveL 1126 to (-20.5, -54.59, -272.44) mm, rotated rx 42.04 ry 15.1 rz 65.25 deg; joints [-19.329, -38.406, 103.053, 141.887, 51.593, -27.708, -175]
  MoveL 1127 to (-22.37, -53.57, -272.62) mm, rotated rx 42.04 ry 15.1 rz 65.25 deg; joints [-19.345, -38.325, 103.095, 141.93, 51.694, -27.798, -175]
  MoveL 1128 to (-24.24, -52.53, -272.71) mm, rotated rx 42.04 ry 15.1 rz 65.25 deg; joints [-19.356, -38.245, 103.14, 141.976, 51.796, -27.891, -175]
  MoveL 1129 to (-25.95, -51.56, -272.92) mm, rotated rx 42.04 ry 15.1 rz 65.25 deg; joints [-19.372, -38.171, 103.18, 142.013, 51.89, -27.974, -175]
  MoveL 1130 to (-28.02, -50.42, -273.07) mm, rotated rx 42.04 ry 15.1 rz 65.25 deg; joints [-19.387, -38.081, 103.227, 142.061, 52.001, -28.074, -175]
  MoveL 1131 to (-30.26, -49.18, -273.19) mm, rotated rx 42.04 ry 15.1 rz 65.25 deg; joints [-19.402, -37.984, 103.278, 142.116, 52.123, -28.184, -175]
  MoveL 1132 to (-32.13, -48.14, -273.19) mm, rotated rx 42.04 ry 15.1 rz 65.25 deg; joints [-19.411, -37.903, 103.323, 142.165, 52.224, -28.278, -175]
  MoveL 1133 to (-33.91, -47.15, -273.26) mm, rotated rx 42.04 ry 15.1 rz 65.25 deg; joints [-19.422, -37.826, 103.365, 142.209, 52.321, -28.366, -175]
  MoveL 1134 to (-35.49, -46.25, -273.44) mm, rotated rx 42.04 ry 15.1 rz 65.25 deg; joints [-19.436, -37.756, 103.401, 142.242, 52.408, -28.442, -175]
  MoveL 1135 to (-37.11, -45.31, -273.65) mm, rotated rx 42.04 ry 15.1 rz 65.25 deg; joints [-19.452, -37.686, 103.438, 142.275, 52.497, -28.519, -175]
  MoveL 1136 to (-39.17, -44.15, -273.78) mm, rotated rx 42.04 ry 15.1 rz 65.25 deg; joints [-19.466, -37.595, 103.484, 142.322, 52.609, -28.618, -175]
  MoveL 1137 to (-41.42, -42.9, -273.89) mm, rotated rx 42.04 ry 15.1 rz 65.25 deg; joints [-19.481, -37.496, 103.535, 142.375, 52.732, -28.727, -175]
  MoveL 1138 to (-45.15, -40.83, -273.89) mm, rotated rx 42.04 ry 15.1 rz 65.25 deg; joints [-19.498, -37.332, 103.62, 142.47, 52.934, -28.911, -175]
  MoveL 1139 to (-45.23, -40.52, -274.59) mm, rotated rx 42.04 ry 15.1 rz 65.25 deg; joints [-19.527, -37.33, 103.629, 142.442, 52.949, -28.908, -175]
  MoveL 1140 to (-44.91, -40.55, -274.93) mm, rotated rx 42.04 ry 15.1 rz 65.25 deg; joints [-19.54, -37.345, 103.626, 142.419, 52.938, -28.889, -175]
  MoveL 1141 to (-44.9, -40.54, -275.15) mm, rotated rx 42.04 ry 15.1 rz 65.25 deg; joints [-19.548, -37.344, 103.622, 142.408, 52.938, -28.883, -175]
  MoveL 1142 to (-45.17, -40.49, -275.26) mm, rotated rx 42.04 ry 15.1 rz 65.25 deg; joints [-19.552, -37.328, 103.617, 142.407, 52.947, -28.889, -175]
  MoveL 1143 to (-45.62, -40.47, -275.29) mm, rotated rx 42.04 ry 15.1 rz 65.25 deg; joints [-19.553, -37.301, 103.607, 142.414, 52.96, -28.902, -175]
  MoveL 1144 to (-46.09, -40.48, -275.32) mm, rotated rx 42.04 ry 15.1 rz 65.25 deg; joints [-19.554, -37.272, 103.593, 142.421, 52.973, -28.914, -175]
  MoveL 1145 to (-46.53, -40.49, -275.36) mm, rotated rx 42.04 ry 15.1 rz 65.25 deg; joints [-19.555, -37.245, 103.58, 142.425, 52.984, -28.924, -175]
  MoveL 1146 to (-46.93, -40.49, -275.43) mm, rotated rx 42.04 ry 15.1 rz 65.25 deg; joints [-19.557, -37.221, 103.568, 142.429, 52.995, -28.933, -175]
  MoveL 1147 to (-47.34, -40.5, -275.49) mm, rotated rx 42.04 ry 15.1 rz 65.25 deg; joints [-19.559, -37.195, 103.556, 142.433, 53.006, -28.942, -175]
  MoveL 1148 to (-47.78, -40.52, -275.53) mm, rotated rx 42.04 ry 15.1 rz 65.25 deg; joints [-19.56, -37.167, 103.542, 142.438, 53.017, -28.952, -175]
  MoveL 1149 to (-48.3, -40.55, -275.55) mm, rotated rx 42.04 ry 15.1 rz 65.25 deg; joints [-19.56, -37.135, 103.525, 142.445, 53.029, -28.964, -175]
  MoveL 1150 to (-48.83, -40.56, -275.62) mm, rotated rx 42.04 ry 15.1 rz 65.25 deg; joints [-19.562, -37.102, 103.509, 142.451, 53.043, -28.976, -175]
  MoveL 1151 to (-49.36, -40.59, -275.65) mm, rotated rx 42.04 ry 15.1 rz 65.25 deg; joints [-19.563, -37.069, 103.492, 142.458, 53.056, -28.988, -175]
  MoveL 1152 to (-49.87, -40.63, -275.65) mm, rotated rx 42.04 ry 15.1 rz 65.25 deg; joints [-19.562, -37.037, 103.475, 142.465, 53.068, -29, -175]
  MoveL 1153 to (-50.39, -40.68, -275.65) mm, rotated rx 42.04 ry 15.1 rz 65.25 deg; joints [-19.561, -37.004, 103.458, 142.474, 53.08, -29.012, -175]
  MoveL 1154 to (-51.08, -40.75, -275.62) mm, rotated rx 42.04 ry 15.1 rz 65.25 deg; joints [-19.558, -36.961, 103.435, 142.486, 53.095, -29.028, -175]
  MoveL 1155 to (-51.74, -40.82, -275.59) mm, rotated rx 42.04 ry 15.1 rz 65.25 deg; joints [-19.556, -36.919, 103.412, 142.497, 53.11, -29.044, -175]
  MoveL 1156 to (-52.34, -40.88, -275.58) mm, rotated rx 42.04 ry 15.1 rz 65.25 deg; joints [-19.555, -36.882, 103.392, 142.507, 53.123, -29.058, -175]
  MoveL 1157 to (-52.81, -40.9, -275.62) mm, rotated rx 42.04 ry 15.1 rz 65.25 deg; joints [-19.556, -36.853, 103.377, 142.512, 53.135, -29.068, -175]
  MoveL 1158 to (-53.22, -40.9, -275.68) mm, rotated rx 42.04 ry 15.1 rz 65.25 deg; joints [-19.557, -36.827, 103.365, 142.516, 53.146, -29.078, -175]
  MoveL 1159 to (-53.63, -40.91, -275.73) mm, rotated rx 42.04 ry 15.1 rz 65.25 deg; joints [-19.559, -36.802, 103.352, 142.52, 53.156, -29.087, -175]
  MoveL 1160 to (-54.07, -40.93, -275.77) mm, rotated rx 42.04 ry 15.1 rz 65.25 deg; joints [-19.56, -36.774, 103.338, 142.525, 53.167, -29.097, -175]
  MoveL 1161 to (-55.64, -41.06, -275.77) mm, rotated rx 42.04 ry 15.1 rz 65.25 deg; joints [-19.557, -36.676, 103.286, 142.549, 53.203, -29.133, -175]
  MoveL 1162 to (-58.53, -41.08, -276.15) mm, rotated rx 42.04 ry 15.1 rz 65.25 deg; joints [-19.569, -36.497, 103.199, 142.578, 53.279, -29.198, -175]
  MoveL 1163 to (-59.77, -40.9, -276.62) mm, rotated rx 42.04 ry 15.1 rz 65.25 deg; joints [-19.587, -36.423, 103.171, 142.578, 53.319, -29.225, -175]
  MoveL 1164 to (-60.87, -40.59, -277.28) mm, rotated rx 42.04 ry 15.1 rz 65.25 deg; joints [-19.613, -36.359, 103.152, 142.567, 53.362, -29.249, -175]
  MoveL 1165 to (-61.83, -40.16, -278.12) mm, rotated rx 42.04 ry 15.1 rz 65.25 deg; joints [-19.648, -36.305, 103.144, 142.548, 53.406, -29.27, -175]
  MoveL 1166 to (-62.66, -39.6, -279.16) mm, rotated rx 42.04 ry 15.1 rz 65.25 deg; joints [-19.692, -36.262, 103.145, 142.518, 53.452, -29.287, -175]
  MoveL 1167 to (-63.91, -38.11, -281.8) mm, rotated rx 42.04 ry 15.1 rz 65.25 deg; joints [-19.803, -36.205, 103.178, 142.43, 53.55, -29.312, -175]
  MoveL 1168 to (-64.37, -36.59, -284.43) mm, rotated rx 42.04 ry 15.1 rz 65.25 deg; joints [-19.916, -36.196, 103.233, 142.329, 53.628, -29.317, -175]
  MoveL 1169 to (-64.21, -35.99, -285.47) mm, rotated rx 42.04 ry 15.1 rz 65.25 deg; joints [-19.961, -36.213, 103.263, 142.284, 53.649, -29.31, -175]
  MoveL 1170 to (-63.79, -35.51, -286.32) mm, rotated rx 42.04 ry 15.1 rz 65.25 deg; joints [-19.998, -36.244, 103.295, 142.242, 53.658, -29.297, -175]
  MoveL 1171 to (-63.11, -35.15, -286.98) mm, rotated rx 42.04 ry 15.1 rz 65.25 deg; joints [-20.026, -36.29, 103.329, 142.204, 53.656, -29.277, -175]
  MoveL 1172 to (-62.17, -34.89, -287.45) mm, rotated rx 42.04 ry 15.1 rz 65.25 deg; joints [-20.047, -36.349, 103.365, 142.169, 53.642, -29.25, -175]
  MoveL 1173 to (-60.97, -34.75, -287.73) mm, rotated rx 42.04 ry 15.1 rz 65.25 deg; joints [-20.06, -36.423, 103.402, 142.137, 53.616, -29.218, -175]
  MoveL 1174 to (-59.51, -34.72, -287.82) mm, rotated rx 42.04 ry 15.1 rz 65.25 deg; joints [-20.065, -36.512, 103.441, 142.109, 53.578, -29.178, -175]
  MoveL 1175 to (-58.99, -34.73, -287.82) mm, rotated rx 42.04 ry 15.1 rz 65.25 deg; joints [-20.066, -36.543, 103.454, 142.101, 53.564, -29.164, -175]
  MoveL 1176 to (-58.52, -34.75, -287.8) mm, rotated rx 42.04 ry 15.1 rz 65.25 deg; joints [-20.065, -36.571, 103.466, 142.094, 53.55, -29.151, -175]
  MoveL 1177 to (-58.12, -34.78, -287.76) mm, rotated rx 42.04 ry 15.1 rz 65.25 deg; joints [-20.063, -36.595, 103.475, 142.089, 53.538, -29.141, -175]
  MoveL 1178 to (-57.73, -34.82, -287.7) mm, rotated rx 42.04 ry 15.1 rz 65.25 deg; joints [-20.061, -36.618, 103.483, 142.085, 53.526, -29.13, -175]
  MoveL 1179 to (-57.3, -34.85, -287.66) mm, rotated rx 42.04 ry 15.1 rz 65.25 deg; joints [-20.06, -36.644, 103.493, 142.079, 53.513, -29.119, -175]
  MoveL 1180 to (-56.81, -34.87, -287.63) mm, rotated rx 42.04 ry 15.1 rz 65.25 deg; joints [-20.059, -36.673, 103.505, 142.072, 53.499, -29.106, -175]
  MoveL 1181 to (-56.29, -34.88, -287.63) mm, rotated rx 42.04 ry 15.1 rz 65.25 deg; joints [-20.059, -36.704, 103.518, 142.063, 53.485, -29.091, -175]
  MoveL 1182 to (-55.82, -34.89, -287.61) mm, rotated rx 42.04 ry 15.1 rz 65.25 deg; joints [-20.059, -36.732, 103.529, 142.056, 53.472, -29.079, -175]
  MoveL 1183 to (-55.42, -34.91, -287.56) mm, rotated rx 42.04 ry 15.1 rz 65.25 deg; joints [-20.057, -36.757, 103.539, 142.052, 53.46, -29.069, -175]
  MoveL 1184 to (-55.03, -34.94, -287.5) mm, rotated rx 42.04 ry 15.1 rz 65.25 deg; joints [-20.055, -36.78, 103.548, 142.048, 53.448, -29.059, -175]
  MoveL 1185 to (-54.6, -34.96, -287.45) mm, rotated rx 42.04 ry 15.1 rz 65.25 deg; joints [-20.053, -36.806, 103.559, 142.043, 53.436, -29.047, -175]
  MoveL 1186 to (-54.11, -34.98, -287.43) mm, rotated rx 42.04 ry 15.1 rz 65.25 deg; joints [-20.053, -36.835, 103.571, 142.036, 53.422, -29.034, -175]
  MoveL 1187 to (-53.58, -34.99, -287.43) mm, rotated rx 42.04 ry 15.1 rz 65.25 deg; joints [-20.053, -36.867, 103.583, 142.027, 53.407, -29.02, -175]
  MoveL 1188 to (-52.6, -35.08, -287.41) mm, rotated rx 42.04 ry 15.1 rz 65.25 deg; joints [-20.052, -36.924, 103.602, 142.01, 53.377, -28.991, -175]
  MoveC 1189 to (-51.23, -35.24, -287.41) mm, rotated rx 42.04 ry 15.1 rz 65.25 deg; joints [-20.052, -37.002, 103.623, 141.984, 53.332, -28.947, -175] to (-49.85, -35.23, -287.41) mm, rotated rx 42.04 ry 15.1 rz 65.25 deg; joints [-20.053, -37.085, 103.659, 141.961, 53.295, -28.91, -175]
  MoveL 1190 to (-49.85, -35.23, -287.4) mm, rotated rx 42.04 ry 15.1 rz 65.25 deg; joints [-20.053, -37.085, 103.659, 141.962, 53.295, -28.911, -175]
  MoveL 1191 to (-49.19, -35.29, -287.38) mm, rotated rx 42.04 ry 15.1 rz 65.25 deg; joints [-20.052, -37.124, 103.672, 141.951, 53.275, -28.891, -175]
  MoveL 1192 to (-48.63, -35.39, -287.35) mm, rotated rx 42.04 ry 15.1 rz 65.25 deg; joints [-20.05, -37.155, 103.678, 141.941, 53.254, -28.872, -175]
  MoveL 1193 to (-48.35, -35.51, -287.26) mm, rotated rx 42.04 ry 15.1 rz 65.25 deg; joints [-20.046, -37.169, 103.678, 141.939, 53.241, -28.863, -175]
  MoveL 1194 to (-48.41, -35.54, -287.06) mm, rotated rx 42.04 ry 15.1 rz 65.25 deg; joints [-20.038, -37.167, 103.678, 141.949, 53.242, -28.868, -175]
  MoveL 1195 to (-48.82, -35.46, -286.75) mm, rotated rx 42.04 ry 15.1 rz 65.25 deg; joints [-20.027, -37.147, 103.683, 141.973, 53.258, -28.891, -175]
  MoveL 1196 to (-49.09, -35.73, -286.13) mm, rotated rx 42.04 ry 15.1 rz 65.25 deg; joints [-20.001, -37.129, 103.667, 142.005, 53.254, -28.903, -175]
  MoveL 1197 to (-47.36, -36.8, -286.12) mm, rotated rx 42.04 ry 15.1 rz 65.25 deg; joints [-19.991, -37.202, 103.619, 141.96, 53.156, -28.813, -175]
  MoveL 1198 to (-45.59, -38, -286.06) mm, rotated rx 42.04 ry 15.1 rz 65.25 deg; joints [-19.978, -37.275, 103.562, 141.914, 53.05, -28.718, -175]
  MoveL 1199 to (-43.73, -39.31, -285.94) mm, rotated rx 42.04 ry 15.1 rz 65.25 deg; joints [-19.962, -37.35, 103.498, 141.869, 52.937, -28.618, -175]
  MoveL 1200 to (-41.9, -40.6, -285.84) mm, rotated rx 42.04 ry 15.1 rz 65.25 deg; joints [-19.947, -37.423, 103.435, 141.823, 52.826, -28.518, -175]
  MoveL 1201 to (-40.14, -41.84, -285.67) mm, rotated rx 42.04 ry 15.1 rz 65.25 deg; joints [-19.929, -37.494, 103.375, 141.782, 52.719, -28.424, -175]
  MoveL 1202 to (-38.56, -42.97, -285.52) mm, rotated rx 42.04 ry 15.1 rz 65.25 deg; joints [-19.914, -37.557, 103.32, 141.744, 52.623, -28.338, -175]
  MoveL 1203 to (-36.86, -44.15, -285.47) mm, rotated rx 42.04 ry 15.1 rz 65.25 deg; joints [-19.901, -37.624, 103.26, 141.698, 52.52, -28.245, -175]
  MoveL 1204 to (-35.1, -45.39, -285.4) mm, rotated rx 42.04 ry 15.1 rz 65.25 deg; joints [-19.888, -37.694, 103.198, 141.651, 52.413, -28.147, -175]
  MoveL 1205 to (-33.17, -46.74, -285.25) mm, rotated rx 42.04 ry 15.1 rz 65.25 deg; joints [-19.87, -37.77, 103.131, 141.603, 52.296, -28.042, -175]
  MoveL 1206 to (-31.63, -47.82, -285.13) mm, rotated rx 42.04 ry 15.1 rz 65.25 deg; joints [-19.856, -37.83, 103.077, 141.564, 52.203, -27.958, -175]
  MoveL 1207 to (-29.67, -49.18, -284.92) mm, rotated rx 42.04 ry 15.1 rz 65.25 deg; joints [-19.836, -37.908, 103.01, 141.518, 52.084, -27.852, -175]
  MoveL 1208 to (-28.13, -50.25, -284.8) mm, rotated rx 42.04 ry 15.1 rz 65.25 deg; joints [-19.823, -37.969, 102.957, 141.478, 51.991, -27.768, -175]
  MoveL 1209 to (-26.37, -51.46, -284.64) mm, rotated rx 42.04 ry 15.1 rz 65.25 deg; joints [-19.806, -38.038, 102.896, 141.434, 51.886, -27.672, -175]
  MoveL 1210 to (-24.41, -52.82, -284.59) mm, rotated rx 42.04 ry 15.1 rz 65.25 deg; joints [-19.792, -38.113, 102.825, 141.378, 51.767, -27.562, -175]
  MoveL 1211 to (-22.86, -53.89, -284.48) mm, rotated rx 42.04 ry 15.1 rz 65.25 deg; joints [-19.779, -38.173, 102.77, 141.338, 51.674, -27.476, -175]
  MoveL 1212 to (-21.1, -55.1, -284.32) mm, rotated rx 42.04 ry 15.1 rz 65.25 deg; joints [-19.762, -38.242, 102.71, 141.293, 51.569, -27.38, -175]
  MoveL 1213 to (-19.14, -56.45, -284.27) mm, rotated rx 42.04 ry 15.1 rz 65.25 deg; joints [-19.748, -38.316, 102.637, 141.236, 51.451, -27.269, -175]
  MoveL 1214 to (-17.59, -57.52, -284.15) mm, rotated rx 42.04 ry 15.1 rz 65.25 deg; joints [-19.735, -38.376, 102.582, 141.194, 51.358, -27.183, -175]
  MoveL 1215 to (-15.75, -58.77, -284.05) mm, rotated rx 42.04 ry 15.1 rz 65.25 deg; joints [-19.72, -38.446, 102.517, 141.143, 51.248, -27.08, -175]
  MoveL 1216 to (-13.92, -60.03, -283.98) mm, rotated rx 42.04 ry 15.1 rz 65.25 deg; joints [-19.707, -38.515, 102.449, 141.09, 51.137, -26.976, -175]
  MoveL 1217 to (-12.35, -61.07, -283.8) mm, rotated rx 42.04 ry 15.1 rz 65.25 deg; joints [-19.691, -38.577, 102.397, 141.051, 51.045, -26.891, -175]
  MoveL 1218 to (-10.89, -62, -283.55) mm, rotated rx 42.04 ry 15.1 rz 65.25 deg; joints [-19.674, -38.635, 102.354, 141.02, 50.961, -26.816, -175]
  MoveL 1219 to (-9.5, -62.85, -283.2) mm, rotated rx 42.04 ry 15.1 rz 65.25 deg; joints [-19.653, -38.693, 102.319, 140.996, 50.883, -26.75, -175]
  MoveL 1220 to (-10.45, -61.68, -282.51) mm, rotated rx 42.04 ry 15.1 rz 65.25 deg; joints [-19.639, -38.681, 102.417, 141.069, 50.965, -26.846, -175]
  MoveL 1221 to (-10.29, -61.84, -282.5) mm, rotated rx 42.04 ry 15.1 rz 65.25 deg; joints [-19.637, -38.686, 102.407, 141.064, 50.953, -26.835, -175]
  MoveL 1222 to (-10.11, -62.08, -282.49) mm, rotated rx 42.04 ry 15.1 rz 65.25 deg; joints [-19.635, -38.689, 102.39, 141.057, 50.937, -26.82, -175]
  MoveL 1223 to (-9.89, -62.49, -282.46) mm, rotated rx 42.04 ry 15.1 rz 65.25 deg; joints [-19.63, -38.689, 102.36, 141.047, 50.912, -26.797, -175]
  MoveL 1224 to (-9.66, -62.97, -282.42) mm, rotated rx 42.04 ry 15.1 rz 65.25 deg; joints [-19.624, -38.688, 102.324, 141.036, 50.883, -26.771, -175]
  MoveL 1225 to (-9.41, -63.53, -282.38) mm, rotated rx 42.04 ry 15.1 rz 65.25 deg; joints [-19.617, -38.685, 102.281, 141.023, 50.849, -26.742, -175]
  MoveL 1226 to (-8.45, -65.97, -282.38) mm, rotated rx 42.04 ry 15.1 rz 65.25 deg; joints [-19.594, -38.664, 102.086, 140.962, 50.708, -26.612, -175]
  MoveL 1227 to (-8.22, -66.53, -282.35) mm, rotated rx 42.04 ry 15.1 rz 65.25 deg; joints [-19.587, -38.66, 102.042, 140.949, 50.675, -26.582, -175]
  MoveL 1228 to (-7.94, -67.16, -282.29) mm, rotated rx 42.04 ry 15.1 rz 65.25 deg; joints [-19.579, -38.657, 101.994, 140.935, 50.638, -26.549, -175]
  MoveL 1229 to (-7.69, -67.74, -282.26) mm, rotated rx 42.04 ry 15.1 rz 65.25 deg; joints [-19.572, -38.653, 101.949, 140.922, 50.604, -26.518, -175]
  MoveL 1230 to (-7.5, -68.22, -282.26) mm, rotated rx 42.04 ry 15.1 rz 65.25 deg; joints [-19.568, -38.648, 101.91, 140.909, 50.576, -26.492, -175]
  MoveL 1231 to (-7.32, -68.68, -282.25) mm, rotated rx 42.04 ry 15.1 rz 65.25 deg; joints [-19.563, -38.644, 101.874, 140.898, 50.55, -26.468, -175]
  MoveL 1232 to (-7.13, -69.17, -282.25) mm, rotated rx 42.04 ry 15.1 rz 65.25 deg; joints [-19.559, -38.64, 101.834, 140.885, 50.522, -26.442, -175]
  MoveL 1233 to (-6.94, -69.65, -282.24) mm, rotated rx 42.04 ry 15.1 rz 65.25 deg; joints [-19.554, -38.635, 101.796, 140.873, 50.494, -26.416, -175]
  MoveL 1234 to (-6.76, -70.09, -282.22) mm, rotated rx 42.04 ry 15.1 rz 65.25 deg; joints [-19.549, -38.632, 101.761, 140.863, 50.468, -26.392, -175]
  MoveL 1235 to (-6.57, -70.52, -282.17) mm, rotated rx 42.04 ry 15.1 rz 65.25 deg; joints [-19.543, -38.63, 101.729, 140.854, 50.443, -26.37, -175]
  MoveL 1236 to (-6.38, -70.98, -282.15) mm, rotated rx 42.04 ry 15.1 rz 65.25 deg; joints [-19.538, -38.626, 101.692, 140.843, 50.416, -26.346, -175]
  MoveL 1237 to (-6.19, -71.47, -282.15) mm, rotated rx 42.04 ry 15.1 rz 65.25 deg; joints [-19.533, -38.622, 101.653, 140.83, 50.388, -26.319, -175]
  MoveL 1238 to (-5.8, -72.45, -282.15) mm, rotated rx 42.04 ry 15.1 rz 65.25 deg; joints [-19.524, -38.612, 101.574, 140.805, 50.331, -26.267, -175]
  Set speed (1000.0 mm/s)
  MoveL 1239 to (-3.92, -93.98, -282.15) mm, rotated rx 42.04 ry 15.1 rz 65.25 deg; joints [-19.319, -38.009, 99.677, 140.355, 49.271, -25.287, -175]
  Print: /'Flow1'
  Set speed (1000.0 mm/s)
  MoveL 1240 to (115.82, 27.66, -72.15) mm, rotated rx -9.61 ry -16.54 rz 125.97 deg; joints [-7.663, -63.141, 109.635, 206.123, 32.592, -123.586, -235]
  Set speed (1000.0 mm/s)
  MoveL 1241 to (75.15, 46.62, -72.15) mm, rotated rx -9.61 ry -16.54 rz 125.97 deg; joints [-7.768, -65.146, 113.572, 204.695, 34.306, -121.967, -235]
  Set speed (100.0 mm/s)
  MoveL 1242 to (9.2, 77.37, -72.15) mm, rotated rx -9.61 ry -16.54 rz 125.97 deg; joints [-7.953, -68.3, 119.737, 202.712, 37.017, -119.702, -235]
  MoveL 1243 to (8.97, 77.84, -72.15) mm, rotated rx -9.61 ry -16.54 rz 125.97 deg; joints [-7.954, -68.336, 119.771, 202.712, 37.014, -119.703, -235]
  MoveL 1244 to (8.63, 78.39, -72.05) mm, rotated rx -9.61 ry -16.54 rz 125.97 deg; joints [-7.951, -68.379, 119.815, 202.716, 37.015, -119.705, -235]
  MoveL 1245 to (8.33, 78.9, -72) mm, rotated rx -9.61 ry -16.54 rz 125.97 deg; joints [-7.95, -68.419, 119.854, 202.718, 37.015, -119.707, -235]
  MoveL 1246 to (8.06, 79.4, -71.98) mm, rotated rx -9.61 ry -16.54 rz 125.97 deg; joints [-7.95, -68.458, 119.89, 202.719, 37.012, -119.708, -235]
  MoveL 1247 to (6.41, 82.67, -71.98) mm, rotated rx -9.61 ry -16.54 rz 125.97 deg; joints [-7.958, -68.712, 120.122, 202.718, 36.99, -119.715, -235]
  MoveL 1248 to (5.81, 83.99, -72.06) mm, rotated rx -9.61 ry -16.54 rz 125.97 deg; joints [-7.965, -68.813, 120.209, 202.714, 36.976, -119.717, -235]
  MoveL 1249 to (5.44, 85.12, -72.33) mm, rotated rx -9.61 ry -16.54 rz 125.97 deg; joints [-7.98, -68.897, 120.272, 202.704, 36.952, -119.717, -235]
  MoveL 1250 to (5.3, 86.06, -72.77) mm, rotated rx -9.61 ry -16.54 rz 125.97 deg; joints [-8.001, -68.964, 120.309, 202.685, 36.921, -119.715, -235]
  MoveL 1251 to (5.32, 86.45, -73.06) mm, rotated rx -9.61 ry -16.54 rz 125.97 deg; joints [-8.014, -68.991, 120.319, 202.674, 36.901, -119.714, -235]
  MoveL 1252 to (5.4, 86.8, -73.4) mm, rotated rx -9.61 ry -16.54 rz 125.97 deg; joints [-8.029, -69.013, 120.322, 202.66, 36.88, -119.712, -235]
  MoveL 1253 to (5.73, 87.36, -74.19) mm, rotated rx -9.61 ry -16.54 rz 125.97 deg; joints [-8.065, -69.045, 120.31, 202.627, 36.831, -119.705, -235]
  MoveL 1254 to (6.29, 87.72, -75.17) mm, rotated rx -9.61 ry -16.54 rz 125.97 deg; joints [-8.108, -69.059, 120.273, 202.588, 36.773, -119.697, -235]
  MoveL 1255 to (8.11, 87.87, -77.66) mm, rotated rx -9.61 ry -16.54 rz 125.97 deg; joints [-8.214, -69.036, 120.125, 202.486, 36.632, -119.674, -235]
  MoveL 1256 to (10.25, 87.29, -80.14) mm, rotated rx -9.61 ry -16.54 rz 125.97 deg; joints [-8.318, -68.956, 119.929, 202.383, 36.5, -119.647, -235]
  MoveL 1257 to (12.1, 86.03, -81.91) mm, rotated rx -9.61 ry -16.54 rz 125.97 deg; joints [-8.391, -68.835, 119.738, 202.306, 36.418, -119.621, -235]
  MoveL 1258 to (12.91, 85.14, -82.54) mm, rotated rx -9.61 ry -16.54 rz 125.97 deg; joints [-8.415, -68.759, 119.644, 202.277, 36.396, -119.608, -235]
  MoveL 1259 to (13.64, 84.08, -82.98) mm, rotated rx -9.61 ry -16.54 rz 125.97 deg; joints [-8.431, -68.672, 119.551, 202.255, 36.386, -119.596, -235]
  MoveL 1260 to (14.89, 81.45, -83.33) mm, rotated rx -9.61 ry -16.54 rz 125.97 deg; joints [-8.44, -68.468, 119.37, 202.23, 36.405, -119.574, -235]
  MoveL 1261 to (15.99, 78.5, -83.34) mm, rotated rx -9.61 ry -16.54 rz 125.97 deg; joints [-8.433, -68.246, 119.192, 202.218, 36.447, -119.552, -235]
  MoveL 1262 to (16.17, 78.04, -83.36) mm, rotated rx -9.61 ry -16.54 rz 125.97 deg; joints [-8.432, -68.212, 119.163, 202.216, 36.453, -119.549, -235]
  MoveL 1263 to (16.35, 77.62, -83.4) mm, rotated rx -9.61 ry -16.54 rz 125.97 deg; joints [-8.433, -68.18, 119.135, 202.213, 36.457, -119.545, -235]
  MoveL 1264 to (16.54, 77.25, -83.46) mm, rotated rx -9.61 ry -16.54 rz 125.97 deg; joints [-8.435, -68.151, 119.109, 202.209, 36.459, -119.542, -235]
  MoveL 1265 to (16.72, 76.84, -83.51) mm, rotated rx -9.61 ry -16.54 rz 125.97 deg; joints [-8.436, -68.119, 119.081, 202.205, 36.462, -119.539, -235]
  MoveL 1266 to (16.92, 76.33, -83.54) mm, rotated rx -9.61 ry -16.54 rz 125.97 deg; joints [-8.436, -68.081, 119.049, 202.202, 36.468, -119.535, -235]
  MoveL 1267 to (17.17, 75.73, -83.57) mm, rotated rx -9.61 ry -16.54 rz 125.97 deg; joints [-8.436, -68.035, 119.011, 202.198, 36.474, -119.53, -235]
  MoveL 1268 to (17.39, 75.22, -83.63) mm, rotated rx -9.61 ry -16.54 rz 125.97 deg; joints [-8.437, -67.996, 118.977, 202.194, 36.479, -119.526, -235]
  MoveL 1269 to (17.59, 74.82, -83.71) mm, rotated rx -9.61 ry -16.54 rz 125.97 deg; joints [-8.439, -67.965, 118.948, 202.189, 36.481, -119.522, -235]
  MoveL 1270 to (17.77, 74.42, -83.76) mm, rotated rx -9.61 ry -16.54 rz 125.97 deg; joints [-8.44, -67.935, 118.922, 202.185, 36.484, -119.518, -235]
  MoveL 1271 to (17.95, 73.98, -83.78) mm, rotated rx -9.61 ry -16.54 rz 125.97 deg; joints [-8.44, -67.901, 118.893, 202.183, 36.489, -119.515, -235]
  MoveL 1272 to (18.13, 73.49, -83.78) mm, rotated rx -9.61 ry -16.54 rz 125.97 deg; joints [-8.439, -67.864, 118.864, 202.181, 36.496, -119.512, -235]
  MoveL 1273 to (18.32, 72.98, -83.78) mm, rotated rx -9.61 ry -16.54 rz 125.97 deg; joints [-8.438, -67.826, 118.833, 202.179, 36.503, -119.508, -235]
  MoveL 1274 to (18.53, 72.45, -83.79) mm, rotated rx -9.61 ry -16.54 rz 125.97 deg; joints [-8.437, -67.786, 118.799, 202.177, 36.509, -119.505, -235]
  MoveL 1275 to (18.79, 71.84, -83.82) mm, rotated rx -9.61 ry -16.54 rz 125.97 deg; joints [-8.437, -67.74, 118.759, 202.174, 36.515, -119.501, -235]
  MoveL 1276 to (19.05, 71.31, -83.89) mm, rotated rx -9.61 ry -16.54 rz 125.97 deg; joints [-8.438, -67.699, 118.721, 202.17, 36.517, -119.498, -235]
  MoveL 1277 to (19.28, 70.92, -83.99) mm, rotated rx -9.61 ry -16.54 rz 125.97 deg; joints [-8.442, -67.668, 118.69, 202.165, 36.517, -119.494, -235]
  MoveL 1278 to (19.27, 70.91, -84.23) mm, rotated rx -9.61 ry -16.54 rz 125.97 deg; joints [-8.452, -67.667, 118.69, 202.148, 36.514, -119.484, -235]
  MoveL 1279 to (19.02, 71.22, -84.58) mm, rotated rx -9.61 ry -16.54 rz 125.97 deg; joints [-8.469, -67.691, 118.717, 202.121, 36.513, -119.466, -235]
  MoveL 1280 to (19.23, 72.04, -85.55) mm, rotated rx -9.61 ry -16.54 rz 125.97 deg; joints [-8.512, -67.742, 118.722, 202.077, 36.461, -119.453, -235]
  MoveL 1281 to (20.95, 70.79, -85.55) mm, rotated rx -9.61 ry -16.54 rz 125.97 deg; joints [-8.505, -67.629, 118.548, 202.118, 36.405, -119.498, -235]
  MoveL 1282 to (22.83, 69.48, -85.68) mm, rotated rx -9.61 ry -16.54 rz 125.97 deg; joints [-8.504, -67.51, 118.36, 202.156, 36.342, -119.543, -235]
  MoveL 1283 to (24.6, 68.21, -85.74) mm, rotated rx -9.61 ry -16.54 rz 125.97 deg; joints [-8.5, -67.395, 118.181, 202.195, 36.284, -119.588, -235]
  MoveL 1284 to (26.34, 66.98, -85.87) mm, rotated rx -9.61 ry -16.54 rz 125.97 deg; joints [-8.499, -67.284, 118.006, 202.229, 36.225, -119.629, -235]
  MoveL 1285 to (28.09, 65.75, -86.02) mm, rotated rx -9.61 ry -16.54 rz 125.97 deg; joints [-8.499, -67.172, 117.83, 202.262, 36.165, -119.67, -235]
  MoveL 1286 to (29.82, 64.51, -86.15) mm, rotated rx -9.61 ry -16.54 rz 125.97 deg; joints [-8.498, -67.06, 117.654, 202.296, 36.107, -119.712, -235]
  MoveL 1287 to (31.56, 63.27, -86.35) mm, rotated rx -9.61 ry -16.54 rz 125.97 deg; joints [-8.501, -66.947, 117.477, 202.326, 36.046, -119.751, -235]
  MoveL 1288 to (33.29, 62.04, -86.47) mm, rotated rx -9.61 ry -16.54 rz 125.97 deg; joints [-8.5, -66.835, 117.301, 202.361, 35.987, -119.794, -235]
  MoveL 1289 to (35.03, 60.78, -86.53) mm, rotated rx -9.61 ry -16.54 rz 125.97 deg; joints [-8.496, -66.722, 117.124, 202.401, 35.929, -119.839, -235]
  MoveL 1290 to (36.78, 59.52, -86.67) mm, rotated rx -9.61 ry -16.54 rz 125.97 deg; joints [-8.495, -66.608, 116.946, 202.436, 35.87, -119.882, -235]
  MoveL 1291 to (38.59, 58.22, -86.85) mm, rotated rx -9.61 ry -16.54 rz 125.97 deg; joints [-8.496, -66.491, 116.761, 202.47, 35.807, -119.924, -235]
  MoveL 1292 to (40.39, 56.91, -87.03) mm, rotated rx -9.61 ry -16.54 rz 125.97 deg; joints [-8.498, -66.373, 116.576, 202.503, 35.745, -119.967, -235]
  MoveL 1293 to (41.91, 55.81, -87.27) mm, rotated rx -9.61 ry -16.54 rz 125.97 deg; joints [-8.502, -66.273, 116.419, 202.526, 35.692, -119.999, -235]
  MoveL 1294 to (44.06, 54.24, -87.38) mm, rotated rx -9.61 ry -16.54 rz 125.97 deg; joints [-8.499, -66.131, 116.198, 202.574, 35.619, -120.055, -235]
  Set speed (1000.0 mm/s)
  MoveL 1295 to (85.12, 35.09, -87.38) mm, rotated rx -9.61 ry -16.54 rz 125.97 deg; joints [-8.367, -64.157, 112.299, 203.882, 33.884, -121.526, -235]
  Set speed (1000.0 mm/s)
  MoveL 1296 to (82.7, 29.9, -99.26) mm, rotated rx -9.61 ry -16.54 rz 125.97 deg; joints [-8.859, -63.812, 112.239, 202.9, 34.015, -120.785, -235]
  Set speed (100.0 mm/s)
  MoveL 1297 to (56.7, 42.02, -99.26) mm, rotated rx -9.61 ry -16.54 rz 125.97 deg; joints [-8.952, -65.059, 114.72, 202.065, 35.132, -119.855, -235]
  MoveL 1298 to (55.46, 43.21, -99.02) mm, rotated rx -9.61 ry -16.54 rz 125.97 deg; joints [-8.947, -65.16, 114.859, 202.052, 35.169, -119.835, -235]
  MoveL 1299 to (53.98, 44.58, -98.95) mm, rotated rx -9.61 ry -16.54 rz 125.97 deg; joints [-8.951, -65.278, 115.023, 202.021, 35.211, -119.801, -235]
  MoveL 1300 to (52.47, 45.98, -98.81) mm, rotated rx -9.61 ry -16.54 rz 125.97 deg; joints [-8.951, -65.397, 115.19, 201.995, 35.255, -119.77, -235]
  MoveL 1301 to (50.68, 47.67, -98.67) mm, rotated rx -9.61 ry -16.54 rz 125.97 deg; joints [-8.953, -65.54, 115.388, 201.963, 35.305, -119.732, -235]
  MoveL 1302 to (49.11, 49.12, -98.67) mm, rotated rx -9.61 ry -16.54 rz 125.97 deg; joints [-8.96, -65.664, 115.56, 201.926, 35.349, -119.693, -235]
  MoveL 1303 to (47.38, 50.72, -98.51) mm, rotated rx -9.61 ry -16.54 rz 125.97 deg; joints [-8.961, -65.8, 115.751, 201.896, 35.399, -119.657, -235]
  MoveL 1304 to (45.92, 52.07, -98.33) mm, rotated rx -9.61 ry -16.54 rz 125.97 deg; joints [-8.96, -65.916, 115.912, 201.875, 35.441, -119.63, -235]
  MoveL 1305 to (44.42, 53.47, -98.24) mm, rotated rx -9.61 ry -16.54 rz 125.97 deg; joints [-8.962, -66.035, 116.076, 201.847, 35.482, -119.598, -235]
  MoveL 1306 to (42.85, 54.91, -98.02) mm, rotated rx -9.61 ry -16.54 rz 125.97 deg; joints [-8.96, -66.159, 116.249, 201.825, 35.528, -119.57, -235]
  MoveL 1307 to (41.29, 56.34, -97.86) mm, rotated rx -9.61 ry -16.54 rz 125.97 deg; joints [-8.96, -66.282, 116.419, 201.8, 35.572, -119.539, -235]
  MoveL 1308 to (39.73, 57.77, -97.75) mm, rotated rx -9.61 ry -16.54 rz 125.97 deg; joints [-8.962, -66.404, 116.589, 201.772, 35.616, -119.507, -235]
  MoveL 1309 to (38.15, 59.21, -97.58) mm, rotated rx -9.61 ry -16.54 rz 125.97 deg; joints [-8.962, -66.528, 116.761, 201.748, 35.661, -119.476, -235]
  MoveL 1310 to (36.58, 60.64, -97.44) mm, rotated rx -9.61 ry -16.54 rz 125.97 deg; joints [-8.963, -66.651, 116.931, 201.722, 35.705, -119.445, -235]
  MoveL 1311 to (34.97, 62.11, -97.38) mm, rotated rx -9.61 ry -16.54 rz 125.97 deg; joints [-8.967, -66.777, 117.105, 201.69, 35.748, -119.41, -235]
  MoveL 1312 to (33.38, 63.53, -97.17) mm, rotated rx -9.61 ry -16.54 rz 125.97 deg; joints [-8.965, -66.9, 117.277, 201.668, 35.794, -119.381, -235]
  MoveL 1313 to (31.81, 64.95, -97.04) mm, rotated rx -9.61 ry -16.54 rz 125.97 deg; joints [-8.967, -67.022, 117.447, 201.642, 35.838, -119.35, -235]
  MoveL 1314 to (30.2, 66.4, -96.92) mm, rotated rx -9.61 ry -16.54 rz 125.97 deg; joints [-8.969, -67.147, 117.619, 201.614, 35.882, -119.318, -235]
  MoveL 1315 to (28.8, 67.49, -96.71) mm, rotated rx -9.61 ry -16.54 rz 125.97 deg; joints [-8.966, -67.244, 117.765, 201.595, 35.927, -119.291, -235]
  MoveL 1316 to (27.56, 68.28, -96.36) mm, rotated rx -9.61 ry -16.54 rz 125.97 deg; joints [-8.955, -67.319, 117.889, 201.586, 35.976, -119.27, -235]
  MoveL 1317 to (26.45, 68.76, -95.83) mm, rotated rx -9.61 ry -16.54 rz 125.97 deg; joints [-8.936, -67.371, 117.994, 201.589, 36.029, -119.256, -235]
  MoveL 1318 to (27.22, 67.43, -94.98) mm, rotated rx -9.61 ry -16.54 rz 125.97 deg; joints [-8.895, -67.27, 117.897, 201.653, 36.042, -119.296, -235]
